LIN {X 0,Y 502.777,Z 286.86,A -85,B 0,C 180,E1 -5904.169,E2 -5904.169} C_VEL
LIN {X 0,Y 502.835,Z 286.849,A -85,B 0,C 180,E1 -5906.993,E2 -5906.993} C_VEL
LIN {X 0,Y 502.818,Z 286.854,A -85,B 0,C 180,E1 -5910.065,E2 -5910.065} C_VEL
LIN {X 0,Y 502.832,Z 286.851,A -85,B 0,C 180,E1 -5912.533,E2 -5912.533} C_VEL
LIN {X 0,Y 502.745,Z 286.865,A -85,B 0,C 180,E1 -5915.32,E2 -5915.32} C_VEL
LIN {X 0,Y 502.634,Z 287.212,A -85,B 0,C 180,E1 -5916.952,E2 -5916.952} C_VEL
LIN {X 0,Y 502.627,Z 289.501,A -85,B 0,C 180,E1 -5919.539,E2 -5919.539} C_VEL
LIN {X 0,Y 502.586,Z 291.79,A -85,B 0,C 180,E1 -5922.083,E2 -5922.083} C_VEL
LIN {X 0,Y 502.483,Z 294.829,A -85,B 0,C 180,E1 -5925.418,E2 -5925.418} C_VEL
LIN {X 0,Y 502.45,Z 295.372,A -85,B 0,C 180,E1 -5925.967,E2 -5925.967} C_VEL
LIN {X 0,Y 504.497,Z 304.103,A -85,B 0,C 180,E1 -5926.262,E2 -5926.262} C_VEL
LIN {X 0,Y 504.385,Z 317.099,A -85,B 0,C 180,E1 -5926.76,E2 -5926.76} C_VEL
LIN {X 0,Y 504.121,Z 329.241,A -85,B 0,C 180,E1 -5927.391,E2 -5927.391} C_VEL
LIN {X 0,Y 503.852,Z 340.243,A -85,B 0,C 180,E1 -5928.127,E2 -5928.127} C_VEL
LIN {X 0,Y 503.535,Z 350.991,A -85,B 0,C 180,E1 -5929.037,E2 -5929.037} C_VEL
LIN {X 0,Y 503.275,Z 359.741,A -85,B 0,C 180,E1 -5929.947,E2 -5929.947} C_VEL
LIN {X 0,Y 503.027,Z 367.754,A -85,B 0,C 180,E1 -5930.957,E2 -5930.957} C_VEL
LIN {X 0,Y 502.758,Z 375.603,A -85,B 0,C 180,E1 -5932.167,E2 -5932.167} C_VEL
LIN {X 0,Y 502.504,Z 382.721,A -85,B 0,C 180,E1 -5933.576,E2 -5933.576} C_VEL
LIN {X 0,Y 502.378,Z 387.441,A -85,B 0,C 180,E1 -5934.783,E2 -5934.783} C_VEL
LIN {X 0,Y 502.368,Z 391.03,A -85,B 0,C 180,E1 -5935.989,E2 -5935.989} C_VEL
LIN {X 0,Y 502.264,Z 392.903,A -85,B 0,C 180,E1 -5936.791,E2 -5936.791} C_VEL
LIN {X 0,Y 502.172,Z 394.318,A -85,B 0,C 180,E1 -5937.594,E2 -5937.594} C_VEL
LIN {X 0,Y 502.095,Z 395.883,A -85,B 0,C 180,E1 -5939.198,E2 -5939.198} C_VEL
LIN {X 0,Y 502.088,Z 396.094,A -85,B 0,C 180,E1 -5940,E2 -5940} C_VEL
LIN {X 0,Y 502.091,Z 395.878,A -85,B 0,C 180,E1 -5940.802,E2 -5940.802} C_VEL
LIN {X 0,Y 502.156,Z 394.273,A -85,B 0,C 180,E1 -5942.406,E2 -5942.406} C_VEL
LIN {X 0,Y 502.257,Z 392.849,A -85,B 0,C 180,E1 -5943.209,E2 -5943.209} C_VEL
LIN {X 0,Y 502.367,Z 389.926,A -85,B 0,C 180,E1 -5944.413,E2 -5944.413} C_VEL
LIN {X 0,Y 502.349,Z 385.983,A -85,B 0,C 180,E1 -5945.62,E2 -5945.62} C_VEL
LIN {X 0,Y 502.56,Z 380.845,A -85,B 0,C 180,E1 -5946.833,E2 -5946.833} C_VEL
LIN {X 0,Y 502.707,Z 374.417,A -85,B 0,C 180,E1 -5948.037,E2 -5948.037} C_VEL
LIN {X 0,Y 502.959,Z 366.358,A -85,B 0,C 180,E1 -5949.247,E2 -5949.247} C_VEL
LIN {X 0,Y 503.228,Z 358.139,A -85,B 0,C 180,E1 -5950.257,E2 -5950.257} C_VEL
LIN {X 0,Y 503.541,Z 348.098,A -85,B 0,C 180,E1 -5951.268,E2 -5951.268} C_VEL
LIN {X 0,Y 503.888,Z 336.424,A -85,B 0,C 180,E1 -5952.198,E2 -5952.198} C_VEL
LIN {X 0,Y 504.152,Z 325.502,A -85,B 0,C 180,E1 -5952.888,E2 -5952.888} C_VEL
LIN {X 0,Y 504.441,Z 314.183,A -85,B 0,C 180,E1 -5953.444,E2 -5953.444} C_VEL
LIN {X 0,Y 504.385,Z 303.242,A -85,B 0,C 180,E1 -5953.856,E2 -5953.856} C_VEL
LIN {X 0,Y 502.24,Z 293.249,A -85,B 0,C 180,E1 -5954.201,E2 -5954.201} C_VEL
LIN {X 0,Y 502.22,Z 290.004,A -85,B 0,C 180,E1 -5957.09,E2 -5957.09} C_VEL
LIN {X 0,Y 502.21,Z 287.179,A -85,B 0,C 180,E1 -5959.625,E2 -5959.625} C_VEL
LIN {X 0,Y 502.509,Z 286.893,A -85,B 0,C 180,E1 -5962.186,E2 -5962.186} C_VEL
LIN {X 0,Y 502.749,Z 286.862,A -85,B 0,C 180,E1 -5964.795,E2 -5964.795} C_VEL
LIN {X 0,Y 502.83,Z 286.845,A -85,B 0,C 180,E1 -5967.467,E2 -5967.467} C_VEL
LIN {X 0,Y 502.811,Z 286.853,A -85,B 0,C 180,E1 -5970.211,E2 -5970.211} C_VEL
LIN {X 0,Y 502.835,Z 286.847,A -85,B 0,C 180,E1 -5973.031,E2 -5973.031} C_VEL
LIN {X 0,Y 502.776,Z 286.855,A -85,B 0,C 180,E1 -5975.951,E2 -5975.951} C_VEL
LIN {X 0,Y 502.805,Z 286.85,A -85,B 0,C 180,E1 -5978.976,E2 -5978.976} C_VEL
LIN {X 0,Y 502.8,Z 286.858,A -85,B 0,C 180,E1 -5982.139,E2 -5982.139} C_VEL
LIN {X 0,Y 502.804,Z 286.852,A -85,B 0,C 180,E1 -5985.468,E2 -5985.468} C_VEL
LIN {X 0,Y 502.823,Z 286.848,A -85,B 0,C 180,E1 -5988.934,E2 -5988.934} C_VEL
LIN {X 0,Y 502.796,Z 286.854,A -85,B 0,C 180,E1 -5992.046,E2 -5992.046} C_VEL
LIN {X 0,Y 502.757,Z 286.857,A -85,B 0,C 180,E1 -5993.311,E2 -5993.311} C_VEL
LIN {X 0,Y 502.063,Z 286.969,A -85,B 0,C 180,E1 -5993.981,E2 -5993.981} C_VEL
LIN {X 0,Y 499.152,Z 287.31,A -85,B 0,C 180,E1 -5995.069,E2 -5995.069} C_VEL
LIN {X 0,Y 496.681,Z 287.621,A -85,B 0,C 180,E1 -5995.941,E2 -5995.941} C_VEL
LIN {X 0,Y 495.581,Z 288.094,A -85,B 0,C 180,E1 -5996.61,E2 -5996.61} C_VEL
LIN {X 0,Y 495.472,Z 288.423,A -85,B 0,C 180,E1 -5996.834,E2 -5996.834} C_VEL
LIN {X 0,Y 495.363,Z 292.704,A -85,B 0,C 180,E1 -5999.286,E2 -5999.286} C_VEL
LIN {X 0,Y 495.342,Z 297.433,A -85,B 0,C 180,E1 -6002.082,E2 -6002.082} C_VEL
LIN {X 0,Y 495.339,Z 302.675,A -85,B 0,C 180,E1 -6005.238,E2 -6005.238} C_VEL
LIN {X 0,Y 495.229,Z 307.861,A -85,B 0,C 180,E1 -6008.347,E2 -6008.347} C_VEL
LIN {X 0,Y 495.203,Z 312.327,A -85,B 0,C 180,E1 -6010.948,E2 -6010.948} C_VEL
LIN {X 0,Y 495.16,Z 316.922,A -85,B 0,C 180,E1 -6013.509,E2 -6013.509} C_VEL
LIN {X 0,Y 495.232,Z 320.815,A -85,B 0,C 180,E1 -6015.581,E2 -6015.581} C_VEL
LIN {X 0,Y 497.789,Z 333.295,A -85,B 0,C 180,E1 -6015.982,E2 -6015.982} C_VEL
LIN {X 0,Y 497.643,Z 345.934,A -85,B 0,C 180,E1 -6016.473,E2 -6016.473} C_VEL
LIN {X 0,Y 497.244,Z 358.46,A -85,B 0,C 180,E1 -6017.141,E2 -6017.141} C_VEL
LIN {X 0,Y 496.901,Z 370.191,A -85,B 0,C 180,E1 -6017.959,E2 -6017.959} C_VEL
LIN {X 0,Y 496.537,Z 380.605,A -85,B 0,C 180,E1 -6018.881,E2 -6018.881} C_VEL
LIN {X 0,Y 496.156,Z 390.869,A -85,B 0,C 180,E1 -6020.007,E2 -6020.007} C_VEL
LIN {X 0,Y 495.79,Z 399.762,A -85,B 0,C 180,E1 -6021.235,E2 -6021.235} C_VEL
LIN {X 0,Y 495.527,Z 406.907,A -85,B 0,C 180,E1 -6022.462,E2 -6022.462} C_VEL
LIN {X 0,Y 495.353,Z 411.752,A -85,B 0,C 180,E1 -6023.483,E2 -6023.483} C_VEL
LIN {X 0,Y 495.141,Z 416.445,A -85,B 0,C 180,E1 -6024.706,E2 -6024.706} C_VEL
LIN {X 0,Y 495.179,Z 420.026,A -85,B 0,C 180,E1 -6025.931,E2 -6025.931} C_VEL
LIN {X 0,Y 495.158,Z 421.873,A -85,B 0,C 180,E1 -6026.745,E2 -6026.745} C_VEL
LIN {X 0,Y 495.064,Z 423.29,A -85,B 0,C 180,E1 -6027.559,E2 -6027.559} C_VEL
LIN {X 0,Y 494.92,Z 424.899,A -85,B 0,C 180,E1 -6029.186,E2 -6029.186} C_VEL
LIN {X 0,Y 494.916,Z 425.136,A -85,B 0,C 180,E1 -6030,E2 -6030} C_VEL
LIN {X 0,Y 494.964,Z 424.371,A -85,B 0,C 180,E1 -6031.627,E2 -6031.627} C_VEL
LIN {X 0,Y 495.158,Z 422.058,A -85,B 0,C 180,E1 -6033.255,E2 -6033.255} C_VEL
LIN {X 0,Y 495.165,Z 419.219,A -85,B 0,C 180,E1 -6034.477,E2 -6034.477} C_VEL
LIN {X 0,Y 495.246,Z 415.36,A -85,B 0,C 180,E1 -6035.701,E2 -6035.701} C_VEL
LIN {X 0,Y 495.413,Z 410.361,A -85,B 0,C 180,E1 -6036.925,E2 -6036.925} C_VEL
LIN {X 0,Y 495.623,Z 404.046,A -85,B 0,C 180,E1 -6038.152,E2 -6038.152} C_VEL
LIN {X 0,Y 495.93,Z 396.197,A -85,B 0,C 180,E1 -6039.379,E2 -6039.379} C_VEL
LIN {X 0,Y 496.263,Z 388.18,A -85,B 0,C 180,E1 -6040.403,E2 -6040.403} C_VEL
LIN {X 0,Y 496.62,Z 378.361,A -85,B 0,C 180,E1 -6041.427,E2 -6041.427} C_VEL
LIN {X 0,Y 496.951,Z 367.1,A -85,B 0,C 180,E1 -6042.366,E2 -6042.366} C_VEL
LIN {X 0,Y 497.291,Z 356.493,A -85,B 0,C 180,E1 -6043.069,E2 -6043.069} C_VEL
LIN {X 0,Y 497.653,Z 344.47,A -85,B 0,C 180,E1 -6043.683,E2 -6043.683} C_VEL
LIN {X 0,Y 497.759,Z 333.262,A -85,B 0,C 180,E1 -6044.11,E2 -6044.11} C_VEL
LIN {X 0,Y 495.244,Z 320.782,A -85,B 0,C 180,E1 -6044.511,E2 -6044.511} C_VEL
LIN {X 0,Y 495.193,Z 314.298,A -85,B 0,C 180,E1 -6048.029,E2 -6048.029} C_VEL
LIN {X 0,Y 495.21,Z 309.511,A -85,B 0,C 180,E1 -6050.781,E2 -6050.781} C_VEL
LIN {X 0,Y 495.272,Z 305.085,A -85,B 0,C 180,E1 -6053.411,E2 -6053.411} C_VEL
LIN {X 0,Y 495.305,Z 300.623,A -85,B 0,C 180,E1 -6056.096,E2 -6056.096} C_VEL
LIN {X 0,Y 495.357,Z 296.067,A -85,B 0,C 180,E1 -6058.841,E2 -6058.841} C_VEL
LIN {X 0,Y 495.435,Z 291.24,A -85,B 0,C 180,E1 -6061.665,E2 -6061.665} C_VEL
LIN {X 0,Y 495.542,Z 287.763,A -85,B 0,C 180,E1 -6063.703,E2 -6063.703} C_VEL
LIN {X 0,Y 495.713,Z 287.74,A -85,B 0,C 180,E1 -6066.087,E2 -6066.087} C_VEL
LIN {X 0,Y 495.766,Z 287.732,A -85,B 0,C 180,E1 -6068.768,E2 -6068.768} C_VEL
LIN {X 0,Y 495.759,Z 287.732,A -85,B 0,C 180,E1 -6071.781,E2 -6071.781} C_VEL
LIN {X 0,Y 495.74,Z 287.737,A -85,B 0,C 180,E1 -6075.141,E2 -6075.141} C_VEL
LIN {X 0,Y 495.759,Z 287.731,A -85,B 0,C 180,E1 -6078.219,E2 -6078.219} C_VEL
LIN {X 0,Y 495.753,Z 287.734,A -85,B 0,C 180,E1 -6081.408,E2 -6081.408} C_VEL
LIN {X 0,Y 495.684,Z 287.74,A -85,B 0,C 180,E1 -6084.457,E2 -6084.457} C_VEL
LIN {X 0,Y 495.498,Z 287.867,A -85,B 0,C 180,E1 -6086.652,E2 -6086.652} C_VEL
LIN {X 0,Y 495.395,Z 292.519,A -85,B 0,C 180,E1 -6089.288,E2 -6089.288} C_VEL
LIN {X 0,Y 495.337,Z 297.457,A -85,B 0,C 180,E1 -6092.081,E2 -6092.081} C_VEL
LIN {X 0,Y 495.352,Z 302.923,A -85,B 0,C 180,E1 -6095.234,E2 -6095.234} C_VEL
LIN {X 0,Y 495.275,Z 308.313,A -85,B 0,C 180,E1 -6098.349,E2 -6098.349} C_VEL
LIN {X 0,Y 495.221,Z 312.805,A -85,B 0,C 180,E1 -6100.949,E2 -6100.949} C_VEL
LIN {X 0,Y 495.191,Z 317.207,A -85,B 0,C 180,E1 -6103.51,E2 -6103.51} C_VEL
LIN {X 0,Y 495.215,Z 321.03,A -85,B 0,C 180,E1 -6105.698,E2 -6105.698} C_VEL
LIN {X 0,Y 497.608,Z 333.51,A -85,B 0,C 180,E1 -6106.107,E2 -6106.107} C_VEL
LIN {X 0,Y 497.316,Z 346.375,A -85,B 0,C 180,E1 -6106.62,E2 -6106.62} C_VEL
LIN {X 0,Y 496.997,Z 358.421,A -85,B 0,C 180,E1 -6107.27,E2 -6107.27} C_VEL
LIN {X 0,Y 496.737,Z 369.713,A -85,B 0,C 180,E1 -6108.058,E2 -6108.058} C_VEL
LIN {X 0,Y 496.369,Z 380.327,A -85,B 0,C 180,E1 -6108.98,E2 -6108.98} C_VEL
LIN {X 0,Y 496.032,Z 389.812,A -85,B 0,C 180,E1 -6110.005,E2 -6110.005} C_VEL
LIN {X 0,Y 495.76,Z 397.6,A -85,B 0,C 180,E1 -6111.029,E2 -6111.029} C_VEL
LIN {X 0,Y 495.515,Z 405.282,A -85,B 0,C 180,E1 -6112.256,E2 -6112.256} C_VEL
LIN {X 0,Y 495.341,Z 411.412,A -85,B 0,C 180,E1 -6113.482,E2 -6113.482} C_VEL
LIN {X 0,Y 495.137,Z 416.249,A -85,B 0,C 180,E1 -6114.706,E2 -6114.706} C_VEL
LIN {X 0,Y 495.177,Z 419.949,A -85,B 0,C 180,E1 -6115.931,E2 -6115.931} C_VEL
LIN {X 0,Y 495.158,Z 421.841,A -85,B 0,C 180,E1 -6116.745,E2 -6116.745} C_VEL
LIN {X 0,Y 495.064,Z 423.311,A -85,B 0,C 180,E1 -6117.559,E2 -6117.559} C_VEL
LIN {X 0,Y 494.966,Z 424.373,A -85,B 0,C 180,E1 -6118.373,E2 -6118.373} C_VEL
LIN {X 0,Y 494.923,Z 425.018,A -85,B 0,C 180,E1 -6119.186,E2 -6119.186} C_VEL
LIN {X 0,Y 494.921,Z 425.259,A -85,B 0,C 180,E1 -6120,E2 -6120} C_VEL
LIN {X 0,Y 494.925,Z 425.103,A -85,B 0,C 180,E1 -6120.814,E2 -6120.814} C_VEL
LIN {X 0,Y 494.967,Z 424.539,A -85,B 0,C 180,E1 -6121.627,E2 -6121.627} C_VEL
LIN {X 0,Y 495.064,Z 423.562,A -85,B 0,C 180,E1 -6122.441,E2 -6122.441} C_VEL
LIN {X 0,Y 495.175,Z 422.178,A -85,B 0,C 180,E1 -6123.255,E2 -6123.255} C_VEL
LIN {X 0,Y 495.17,Z 419.287,A -85,B 0,C 180,E1 -6124.477,E2 -6124.477} C_VEL
LIN {X 0,Y 495.244,Z 415.341,A -85,B 0,C 180,E1 -6125.701,E2 -6125.701} C_VEL
LIN {X 0,Y 495.429,Z 409.348,A -85,B 0,C 180,E1 -6127.11,E2 -6127.11} C_VEL
LIN {X 0,Y 495.619,Z 402.561,A -85,B 0,C 180,E1 -6128.357,E2 -6128.357} C_VEL
LIN {X 0,Y 495.906,Z 394.128,A -85,B 0,C 180,E1 -6129.586,E2 -6129.586} C_VEL
LIN {X 0,Y 496.177,Z 385.491,A -85,B 0,C 180,E1 -6130.611,E2 -6130.611} C_VEL
LIN {X 0,Y 496.548,Z 375.98,A -85,B 0,C 180,E1 -6131.532,E2 -6131.532} C_VEL
LIN {X 0,Y 496.83,Z 364.145,A -85,B 0,C 180,E1 -6132.454,E2 -6132.454} C_VEL
LIN {X 0,Y 497.158,Z 352.181,A -85,B 0,C 180,E1 -6133.176,E2 -6133.176} C_VEL
LIN {X 0,Y 497.488,Z 339.805,A -85,B 0,C 180,E1 -6133.74,E2 -6133.74} C_VEL
LIN {X 0,Y 497.391,Z 332.518,A -85,B 0,C 180,E1 -6134.003,E2 -6134.003} C_VEL
LIN {X 0,Y 495.304,Z 322.078,A -85,B 0,C 180,E1 -6134.351,E2 -6134.351} C_VEL
LIN {X 0,Y 495.29,Z 316.855,A -85,B 0,C 180,E1 -6137.337,E2 -6137.337} C_VEL
LIN {X 0,Y 495.354,Z 310.64,A -85,B 0,C 180,E1 -6140.775,E2 -6140.775} C_VEL
LIN {X 0,Y 495.347,Z 305.658,A -85,B 0,C 180,E1 -6143.407,E2 -6143.407} C_VEL
LIN {X 0,Y 495.289,Z 300.342,A -85,B 0,C 180,E1 -6146.096,E2 -6146.096} C_VEL
LIN {X 0,Y 495.306,Z 294.597,A -85,B 0,C 180,E1 -6148.845,E2 -6148.845} C_VEL
LIN {X 0,Y 495.282,Z 287.796,A -85,B 0,C 180,E1 -6151.79,E2 -6151.79} C_VEL
LIN {X 0,Y 495.729,Z 287.737,A -85,B 0,C 180,E1 -6154.547,E2 -6154.547} C_VEL
LIN {X 0,Y 495.731,Z 287.737,A -85,B 0,C 180,E1 -6157.562,E2 -6157.562} C_VEL
LIN {X 0,Y 495.761,Z 287.732,A -85,B 0,C 180,E1 -6160.047,E2 -6160.047} C_VEL
LIN {X 0,Y 495.719,Z 287.739,A -85,B 0,C 180,E1 -6162.884,E2 -6162.884} C_VEL
LIN {X 0,Y 495.733,Z 287.735,A -85,B 0,C 180,E1 -6165.999,E2 -6165.999} C_VEL
LIN {X 0,Y 495.764,Z 287.734,A -85,B 0,C 180,E1 -6169.3,E2 -6169.3} C_VEL
LIN {X 0,Y 495.784,Z 287.81,A -85,B 0,C 180,E1 -6169.75,E2 -6169.75} C_VEL
LIN {X 0,Y 497.3,Z 295.706,A -85,B 0,C 180,E1 -6172.577,E2 -6172.577} C_VEL
LIN {X 0,Y 497.951,Z 300.349,A -85,B 0,C 180,E1 -6174.146,E2 -6174.146} C_VEL
LIN {X 0,Y 497.582,Z 308.259,A -85,B 0,C 180,E1 -6176.575,E2 -6176.575} C_VEL
LIN {X 0,Y 497.24,Z 318.209,A -85,B 0,C 180,E1 -6179.562,E2 -6179.562} C_VEL
LIN {X 0,Y 496.824,Z 328.593,A -85,B 0,C 180,E1 -6182.63,E2 -6182.63} C_VEL
LIN {X 0,Y 496.528,Z 339.673,A -85,B 0,C 180,E1 -6185.765,E2 -6185.765} C_VEL
LIN {X 0,Y 496.175,Z 350.733,A -85,B 0,C 180,E1 -6188.827,E2 -6188.827} C_VEL
LIN {X 0,Y 495.884,Z 361.475,A -85,B 0,C 180,E1 -6191.832,E2 -6191.832} C_VEL
LIN {X 0,Y 495.547,Z 372.718,A -85,B 0,C 180,E1 -6194.926,E2 -6194.926} C_VEL
LIN {X 0,Y 495.535,Z 374.712,A -85,B 0,C 180,E1 -6195.472,E2 -6195.472} C_VEL
LIN {X 0,Y 497.769,Z 388.179,A -85,B 0,C 180,E1 -6195.851,E2 -6195.851} C_VEL
LIN {X 0,Y 497.547,Z 400.981,A -85,B 0,C 180,E1 -6196.314,E2 -6196.314} C_VEL
LIN {X 0,Y 497.165,Z 413.171,A -85,B 0,C 180,E1 -6196.928,E2 -6196.928} C_VEL
LIN {X 0,Y 496.815,Z 423.896,A -85,B 0,C 180,E1 -6197.625,E2 -6197.625} C_VEL
LIN {X 0,Y 496.472,Z 434.263,A -85,B 0,C 180,E1 -6198.466,E2 -6198.466} C_VEL
LIN {X 0,Y 496.068,Z 443.539,A -85,B 0,C 180,E1 -6199.387,E2 -6199.387} C_VEL
LIN {X 0,Y 495.791,Z 451.992,A -85,B 0,C 180,E1 -6200.412,E2 -6200.412} C_VEL
LIN {X 0,Y 495.485,Z 460.236,A -85,B 0,C 180,E1 -6201.64,E2 -6201.64} C_VEL
LIN {X 0,Y 495.261,Z 466.876,A -85,B 0,C 180,E1 -6202.868,E2 -6202.868} C_VEL
LIN {X 0,Y 495.178,Z 472.95,A -85,B 0,C 180,E1 -6204.298,E2 -6204.298} C_VEL
LIN {X 0,Y 495.029,Z 476.895,A -85,B 0,C 180,E1 -6205.522,E2 -6205.522} C_VEL
LIN {X 0,Y 495.043,Z 479.807,A -85,B 0,C 180,E1 -6206.745,E2 -6206.745} C_VEL
LIN {X 0,Y 494.961,Z 482.183,A -85,B 0,C 180,E1 -6208.373,E2 -6208.373} C_VEL
LIN {X 0,Y 494.898,Z 483,A -85,B 0,C 180,E1 -6210,E2 -6210} C_VEL
LIN {X 0,Y 494.961,Z 482.184,A -85,B 0,C 180,E1 -6211.627,E2 -6211.627} C_VEL
LIN {X 0,Y 495.043,Z 479.81,A -85,B 0,C 180,E1 -6213.255,E2 -6213.255} C_VEL
LIN {X 0,Y 495.029,Z 476.895,A -85,B 0,C 180,E1 -6214.478,E2 -6214.478} C_VEL
LIN {X 0,Y 495.211,Z 471.802,A -85,B 0,C 180,E1 -6215.999,E2 -6215.999} C_VEL
LIN {X 0,Y 495.277,Z 465.869,A -85,B 0,C 180,E1 -6217.337,E2 -6217.337} C_VEL
LIN {X 0,Y 495.557,Z 459.003,A -85,B 0,C 180,E1 -6218.564,E2 -6218.564} C_VEL
LIN {X 0,Y 495.852,Z 450.412,A -85,B 0,C 180,E1 -6219.793,E2 -6219.793} C_VEL
LIN {X 0,Y 496.183,Z 441.598,A -85,B 0,C 180,E1 -6220.817,E2 -6220.817} C_VEL
LIN {X 0,Y 496.58,Z 430.744,A -85,B 0,C 180,E1 -6221.842,E2 -6221.842} C_VEL
LIN {X 0,Y 496.897,Z 420.211,A -85,B 0,C 180,E1 -6222.636,E2 -6222.636} C_VEL
LIN {X 0,Y 497.282,Z 407.499,A -85,B 0,C 180,E1 -6223.381,E2 -6223.381} C_VEL
LIN {X 0,Y 497.7,Z 394.49,A -85,B 0,C 180,E1 -6223.942,E2 -6223.942} C_VEL
LIN {X 0,Y 497.577,Z 386.8,A -85,B 0,C 180,E1 -6224.193,E2 -6224.193} C_VEL
LIN {X 0,Y 495.543,Z 374.64,A -85,B 0,C 180,E1 -6224.548,E2 -6224.548} C_VEL
LIN {X 0,Y 495.856,Z 363.009,A -85,B 0,C 180,E1 -6227.742,E2 -6227.742} C_VEL
LIN {X 0,Y 496.137,Z 352.111,A -85,B 0,C 180,E1 -6230.784,E2 -6230.784} C_VEL
LIN {X 0,Y 496.412,Z 342.767,A -85,B 0,C 180,E1 -6233.354,E2 -6233.354} C_VEL
LIN {X 0,Y 496.673,Z 331.1,A -85,B 0,C 180,E1 -6236.47,E2 -6236.47} C_VEL
LIN {X 0,Y 496.961,Z 319.522,A -85,B 0,C 180,E1 -6239.668,E2 -6239.668} C_VEL
LIN {X 0,Y 497.19,Z 309.679,A -85,B 0,C 180,E1 -6242.49,E2 -6242.49} C_VEL
LIN {X 0,Y 497.493,Z 301.516,A -85,B 0,C 180,E1 -6244.979,E2 -6244.979} C_VEL
LIN {X 0,Y 497.496,Z 297.199,A -85,B 0,C 180,E1 -6246.393,E2 -6246.393} C_VEL
LIN {X 0,Y 496.317,Z 290.614,A -85,B 0,C 180,E1 -6248.847,E2 -6248.847} C_VEL
LIN {X 0,Y 495.744,Z 287.736,A -85,B 0,C 180,E1 -6250.1,E2 -6250.1} C_VEL
LIN {X 0,Y 495.706,Z 287.742,A -85,B 0,C 180,E1 -6252.886,E2 -6252.886} C_VEL
LIN {X 0,Y 495.727,Z 287.737,A -85,B 0,C 180,E1 -6255.998,E2 -6255.998} C_VEL
LIN {X 0,Y 495.742,Z 287.736,A -85,B 0,C 180,E1 -6258.709,E2 -6258.709} C_VEL
LIN {X 0,Y 495.753,Z 287.732,A -85,B 0,C 180,E1 -6261.408,E2 -6261.408} C_VEL
LIN {X 0,Y 495.751,Z 287.734,A -85,B 0,C 180,E1 -6264.462,E2 -6264.462} C_VEL
LIN {X 0,Y 495.77,Z 287.732,A -85,B 0,C 180,E1 -6267.406,E2 -6267.406} C_VEL
LIN {X 0,Y 495.769,Z 287.731,A -85,B 0,C 180,E1 -6270.254,E2 -6270.254} C_VEL
LIN {X 0,Y 495.809,Z 287.729,A -85,B 0,C 180,E1 -6273.255,E2 -6273.255} C_VEL
LIN {X 0,Y 495.656,Z 287.748,A -85,B 0,C 180,E1 -6275.72,E2 -6275.72} C_VEL
LIN {X 0,Y 495.602,Z 287.999,A -85,B 0,C 180,E1 -6276.605,E2 -6276.605} C_VEL
LIN {X 0,Y 495.608,Z 290.421,A -85,B 0,C 180,E1 -6279.377,E2 -6279.377} C_VEL
LIN {X 0,Y 495.547,Z 292.621,A -85,B 0,C 180,E1 -6281.845,E2 -6281.845} C_VEL
LIN {X 0,Y 495.458,Z 295.66,A -85,B 0,C 180,E1 -6285.207,E2 -6285.207} C_VEL
LIN {X 0,Y 495.468,Z 296.302,A -85,B 0,C 180,E1 -6285.784,E2 -6285.784} C_VEL
LIN {X 0,Y 497.681,Z 305.565,A -85,B 0,C 180,E1 -6286.11,E2 -6286.11} C_VEL
LIN {X 0,Y 497.47,Z 318.582,A -85,B 0,C 180,E1 -6286.624,E2 -6286.624} C_VEL
LIN {X 0,Y 497.215,Z 330.124,A -85,B 0,C 180,E1 -6287.239,E2 -6287.239} C_VEL
LIN {X 0,Y 496.941,Z 340.736,A -85,B 0,C 180,E1 -6287.96,E2 -6287.96} C_VEL
LIN {X 0,Y 496.605,Z 351.541,A -85,B 0,C 180,E1 -6288.882,E2 -6288.882} C_VEL
LIN {X 0,Y 496.326,Z 360.324,A -85,B 0,C 180,E1 -6289.805,E2 -6289.805} C_VEL
LIN {X 0,Y 495.998,Z 369.834,A -85,B 0,C 180,E1 -6291.033,E2 -6291.033} C_VEL
LIN {X 0,Y 495.72,Z 377.365,A -85,B 0,C 180,E1 -6292.26,E2 -6292.26} C_VEL
LIN {X 0,Y 495.483,Z 383.385,A -85,B 0,C 180,E1 -6293.484,E2 -6293.484} C_VEL
LIN {X 0,Y 495.354,Z 388.122,A -85,B 0,C 180,E1 -6294.709,E2 -6294.709} C_VEL
LIN {X 0,Y 495.333,Z 391.725,A -85,B 0,C 180,E1 -6295.932,E2 -6295.932} C_VEL
LIN {X 0,Y 495.213,Z 393.594,A -85,B 0,C 180,E1 -6296.746,E2 -6296.746} C_VEL
LIN {X 0,Y 495.112,Z 395.01,A -85,B 0,C 180,E1 -6297.559,E2 -6297.559} C_VEL
LIN {X 0,Y 495.03,Z 396.572,A -85,B 0,C 180,E1 -6299.187,E2 -6299.187} C_VEL
LIN {X 0,Y 495.022,Z 396.778,A -85,B 0,C 180,E1 -6300,E2 -6300} C_VEL
LIN {X 0,Y 495.026,Z 396.565,A -85,B 0,C 180,E1 -6300.814,E2 -6300.814} C_VEL
LIN {X 0,Y 495.092,Z 394.927,A -85,B 0,C 180,E1 -6302.441,E2 -6302.441} C_VEL
LIN {X 0,Y 495.207,Z 393.501,A -85,B 0,C 180,E1 -6303.254,E2 -6303.254} C_VEL
LIN {X 0,Y 495.331,Z 390.553,A -85,B 0,C 180,E1 -6304.476,E2 -6304.476} C_VEL
LIN {X 0,Y 495.307,Z 386.582,A -85,B 0,C 180,E1 -6305.7,E2 -6305.7} C_VEL
LIN {X 0,Y 495.535,Z 380.533,A -85,B 0,C 180,E1 -6307.108,E2 -6307.108} C_VEL
LIN {X 0,Y 495.751,Z 373.703,A -85,B 0,C 180,E1 -6308.355,E2 -6308.355} C_VEL
LIN {X 0,Y 495.991,Z 365.357,A -85,B 0,C 180,E1 -6309.584,E2 -6309.584} C_VEL
LIN {X 0,Y 496.341,Z 356.757,A -85,B 0,C 180,E1 -6310.607,E2 -6310.607} C_VEL
LIN {X 0,Y 496.69,Z 346.13,A -85,B 0,C 180,E1 -6311.633,E2 -6311.633} C_VEL
LIN {X 0,Y 497.022,Z 335.494,A -85,B 0,C 180,E1 -6312.459,E2 -6312.459} C_VEL
LIN {X 0,Y 497.304,Z 323.908,A -85,B 0,C 180,E1 -6313.172,E2 -6313.172} C_VEL
LIN {X 0,Y 497.613,Z 310.599,A -85,B 0,C 180,E1 -6313.788,E2 -6313.788} C_VEL
LIN {X 0,Y 497.471,Z 304.1,A -85,B 0,C 180,E1 -6314.027,E2 -6314.027} C_VEL
LIN {X 0,Y 495.199,Z 293.764,A -85,B 0,C 180,E1 -6314.381,E2 -6314.381} C_VEL
LIN {X 0,Y 495.148,Z 290.426,A -85,B 0,C 180,E1 -6317.342,E2 -6317.342} C_VEL
LIN {X 0,Y 495.159,Z 288.508,A -85,B 0,C 180,E1 -6319.053,E2 -6319.053} C_VEL
LIN {X 0,Y 495.168,Z 287.809,A -85,B 0,C 180,E1 -6319.916,E2 -6319.916} C_VEL
LIN {X 0,Y 495.509,Z 287.765,A -85,B 0,C 180,E1 -6322.791,E2 -6322.791} C_VEL
LIN {X 0,Y 495.719,Z 287.733,A -85,B 0,C 180,E1 -6325.171,E2 -6325.171} C_VEL
LIN {X 0,Y 495.78,Z 287.724,A -85,B 0,C 180,E1 -6327.891,E2 -6327.891} C_VEL
LIN {X 0,Y 495.753,Z 287.73,A -85,B 0,C 180,E1 -6330.687,E2 -6330.687} C_VEL
LIN {X 0,Y 495.762,Z 287.728,A -85,B 0,C 180,E1 -6333.564,E2 -6333.564} C_VEL
LIN {X 0,Y 495.731,Z 287.736,A -85,B 0,C 180,E1 -6336.544,E2 -6336.544} C_VEL
LIN {X 0,Y 495.76,Z 287.729,A -85,B 0,C 180,E1 -6339.638,E2 -6339.638} C_VEL
LIN {X 0,Y 495.741,Z 287.733,A -85,B 0,C 180,E1 -6342.507,E2 -6342.507} C_VEL
LIN {X 0,Y 495.753,Z 287.728,A -85,B 0,C 180,E1 -6345.139,E2 -6345.139} C_VEL
LIN {X 0,Y 495.76,Z 287.73,A -85,B 0,C 180,E1 -6348.219,E2 -6348.219} C_VEL
LIN {X 0,Y 495.753,Z 287.734,A -85,B 0,C 180,E1 -6351.408,E2 -6351.408} C_VEL
LIN {X 0,Y 495.713,Z 287.736,A -85,B 0,C 180,E1 -6354.459,E2 -6354.459} C_VEL
LIN {X 0,Y 495.539,Z 287.88,A -85,B 0,C 180,E1 -6356.536,E2 -6356.536} C_VEL
LIN {X 0,Y 495.472,Z 288.423,A -85,B 0,C 180,E1 -6356.834,E2 -6356.834} C_VEL
LIN {X 0,Y 494.742,Z 289.665,A -85,B 0,C 180,E1 -6357.497,E2 -6357.497} C_VEL
LIN {X 0,Y 491.823,Z 291.856,A -85,B 0,C 180,E1 -6358.567,E2 -6358.567} C_VEL
LIN {X 0,Y 489.391,Z 293.605,A -85,B 0,C 180,E1 -6359.43,E2 -6359.43} C_VEL
LIN {X 0,Y 488.357,Z 294.856,A -85,B 0,C 180,E1 -6360.099,E2 -6360.099} C_VEL
LIN {X 0,Y 488.276,Z 295.241,A -85,B 0,C 180,E1 -6360.327,E2 -6360.327} C_VEL
LIN {X 0,Y 488.257,Z 298.982,A -85,B 0,C 180,E1 -6362.573,E2 -6362.573} C_VEL
LIN {X 0,Y 488.272,Z 303.531,A -85,B 0,C 180,E1 -6365.328,E2 -6365.328} C_VEL
LIN {X 0,Y 488.168,Z 308.009,A -85,B 0,C 180,E1 -6368.018,E2 -6368.018} C_VEL
LIN {X 0,Y 488.133,Z 312.516,A -85,B 0,C 180,E1 -6370.661,E2 -6370.661} C_VEL
LIN {X 0,Y 488.096,Z 317.167,A -85,B 0,C 180,E1 -6373.263,E2 -6373.263} C_VEL
LIN {X 0,Y 488.184,Z 321.174,A -85,B 0,C 180,E1 -6375.368,E2 -6375.368} C_VEL
LIN {X 0,Y 490.953,Z 334.514,A -85,B 0,C 180,E1 -6375.81,E2 -6375.81} C_VEL
LIN {X 0,Y 490.715,Z 347.401,A -85,B 0,C 180,E1 -6376.331,E2 -6376.331} C_VEL
LIN {X 0,Y 490.337,Z 359.136,A -85,B 0,C 180,E1 -6376.974,E2 -6376.974} C_VEL
LIN {X 0,Y 489.975,Z 370.601,A -85,B 0,C 180,E1 -6377.786,E2 -6377.786} C_VEL
LIN {X 0,Y 489.594,Z 381.016,A -85,B 0,C 180,E1 -6378.721,E2 -6378.721} C_VEL
LIN {X 0,Y 489.188,Z 391.281,A -85,B 0,C 180,E1 -6379.864,E2 -6379.864} C_VEL
LIN {X 0,Y 488.791,Z 400.175,A -85,B 0,C 180,E1 -6381.108,E2 -6381.108} C_VEL
LIN {X 0,Y 488.512,Z 407.32,A -85,B 0,C 180,E1 -6382.353,E2 -6382.353} C_VEL
LIN {X 0,Y 488.311,Z 412.166,A -85,B 0,C 180,E1 -6383.388,E2 -6383.388} C_VEL
LIN {X 0,Y 488.085,Z 416.86,A -85,B 0,C 180,E1 -6384.63,E2 -6384.63} C_VEL
LIN {X 0,Y 488.12,Z 420.44,A -85,B 0,C 180,E1 -6385.872,E2 -6385.872} C_VEL
LIN {X 0,Y 488.077,Z 422.289,A -85,B 0,C 180,E1 -6386.698,E2 -6386.698} C_VEL
LIN {X 0,Y 488.003,Z 423.704,A -85,B 0,C 180,E1 -6387.524,E2 -6387.524} C_VEL
LIN {X 0,Y 487.842,Z 425.314,A -85,B 0,C 180,E1 -6389.175,E2 -6389.175} C_VEL
LIN {X 0,Y 487.836,Z 425.55,A -85,B 0,C 180,E1 -6390,E2 -6390} C_VEL
LIN {X 0,Y 487.894,Z 424.784,A -85,B 0,C 180,E1 -6391.651,E2 -6391.651} C_VEL
LIN {X 0,Y 488.003,Z 423.822,A -85,B 0,C 180,E1 -6392.476,E2 -6392.476} C_VEL
LIN {X 0,Y 488.076,Z 422.471,A -85,B 0,C 180,E1 -6393.302,E2 -6393.302} C_VEL
LIN {X 0,Y 488.099,Z 419.631,A -85,B 0,C 180,E1 -6394.542,E2 -6394.542} C_VEL
LIN {X 0,Y 488.199,Z 415.769,A -85,B 0,C 180,E1 -6395.784,E2 -6395.784} C_VEL
LIN {X 0,Y 488.381,Z 410.769,A -85,B 0,C 180,E1 -6397.026,E2 -6397.026} C_VEL
LIN {X 0,Y 488.593,Z 404.453,A -85,B 0,C 180,E1 -6398.27,E2 -6398.27} C_VEL
LIN {X 0,Y 488.925,Z 396.601,A -85,B 0,C 180,E1 -6399.515,E2 -6399.515} C_VEL
LIN {X 0,Y 489.31,Z 388.58,A -85,B 0,C 180,E1 -6400.552,E2 -6400.552} C_VEL
LIN {X 0,Y 489.676,Z 378.758,A -85,B 0,C 180,E1 -6401.592,E2 -6401.592} C_VEL
LIN {X 0,Y 490.03,Z 367.68,A -85,B 0,C 180,E1 -6402.529,E2 -6402.529} C_VEL
LIN {X 0,Y 490.414,Z 356.878,A -85,B 0,C 180,E1 -6403.255,E2 -6403.255} C_VEL
LIN {X 0,Y 490.79,Z 344.838,A -85,B 0,C 180,E1 -6403.878,E2 -6403.878} C_VEL
LIN {X 0,Y 490.837,Z 334.028,A -85,B 0,C 180,E1 -6404.3,E2 -6404.3} C_VEL
LIN {X 0,Y 488.189,Z 321.092,A -85,B 0,C 180,E1 -6404.725,E2 -6404.725} C_VEL
LIN {X 0,Y 488.116,Z 314.784,A -85,B 0,C 180,E1 -6408.142,E2 -6408.142} C_VEL
LIN {X 0,Y 488.162,Z 309.67,A -85,B 0,C 180,E1 -6411.095,E2 -6411.095} C_VEL
LIN {X 0,Y 488.214,Z 305.189,A -85,B 0,C 180,E1 -6413.77,E2 -6413.77} C_VEL
LIN {X 0,Y 488.273,Z 300.671,A -85,B 0,C 180,E1 -6416.5,E2 -6416.5} C_VEL
LIN {X 0,Y 488.288,Z 296.043,A -85,B 0,C 180,E1 -6419.299,E2 -6419.299} C_VEL
LIN {X 0,Y 488.37,Z 291.119,A -85,B 0,C 180,E1 -6422.172,E2 -6422.172} C_VEL
LIN {X 0,Y 488.48,Z 288.643,A -85,B 0,C 180,E1 -6423.6,E2 -6423.6} C_VEL
LIN {X 0,Y 488.67,Z 288.617,A -85,B 0,C 180,E1 -6426.133,E2 -6426.133} C_VEL
LIN {X 0,Y 488.704,Z 288.611,A -85,B 0,C 180,E1 -6429.254,E2 -6429.254} C_VEL
LIN {X 0,Y 488.71,Z 288.61,A -85,B 0,C 180,E1 -6431.6,E2 -6431.6} C_VEL
LIN {X 0,Y 488.704,Z 288.613,A -85,B 0,C 180,E1 -6434.803,E2 -6434.803} C_VEL
LIN {X 0,Y 488.694,Z 288.615,A -85,B 0,C 180,E1 -6437.474,E2 -6437.474} C_VEL
LIN {X 0,Y 488.736,Z 288.606,A -85,B 0,C 180,E1 -6439.677,E2 -6439.677} C_VEL
LIN {X 0,Y 488.672,Z 288.617,A -85,B 0,C 180,E1 -6442.84,E2 -6442.84} C_VEL
LIN {X 0,Y 488.546,Z 288.631,A -85,B 0,C 180,E1 -6445.872,E2 -6445.872} C_VEL
LIN {X 0,Y 488.419,Z 288.817,A -85,B 0,C 180,E1 -6446.746,E2 -6446.746} C_VEL
LIN {X 0,Y 488.336,Z 294.116,A -85,B 0,C 180,E1 -6449.754,E2 -6449.754} C_VEL
LIN {X 0,Y 488.256,Z 299.044,A -85,B 0,C 180,E1 -6452.573,E2 -6452.573} C_VEL
LIN {X 0,Y 488.288,Z 303.819,A -85,B 0,C 180,E1 -6455.329,E2 -6455.329} C_VEL
LIN {X 0,Y 488.201,Z 308.445,A -85,B 0,C 180,E1 -6458.02,E2 -6458.02} C_VEL
LIN {X 0,Y 488.161,Z 312.971,A -85,B 0,C 180,E1 -6460.663,E2 -6460.663} C_VEL
LIN {X 0,Y 488.123,Z 317.451,A -85,B 0,C 180,E1 -6463.264,E2 -6463.264} C_VEL
LIN {X 0,Y 488.172,Z 321.316,A -85,B 0,C 180,E1 -6465.501,E2 -6465.501} C_VEL
LIN {X 0,Y 490.69,Z 334.833,A -85,B 0,C 180,E1 -6465.96,E2 -6465.96} C_VEL
LIN {X 0,Y 490.371,Z 347.453,A -85,B 0,C 180,E1 -6466.48,E2 -6466.48} C_VEL
LIN {X 0,Y 490.026,Z 359.513,A -85,B 0,C 180,E1 -6467.152,E2 -6467.152} C_VEL
LIN {X 0,Y 489.76,Z 371.161,A -85,B 0,C 180,E1 -6467.99,E2 -6467.99} C_VEL
LIN {X 0,Y 489.364,Z 381.543,A -85,B 0,C 180,E1 -6468.925,E2 -6468.925} C_VEL
LIN {X 0,Y 488.967,Z 391.761,A -85,B 0,C 180,E1 -6470.068,E2 -6470.068} C_VEL
LIN {X 0,Y 488.637,Z 400.661,A -85,B 0,C 180,E1 -6471.314,E2 -6471.314} C_VEL
LIN {X 0,Y 488.421,Z 407.805,A -85,B 0,C 180,E1 -6472.559,E2 -6472.559} C_VEL
LIN {X 0,Y 488.276,Z 413.524,A -85,B 0,C 180,E1 -6473.803,E2 -6473.803} C_VEL
LIN {X 0,Y 488.036,Z 417.997,A -85,B 0,C 180,E1 -6475.043,E2 -6475.043} C_VEL
LIN {X 0,Y 488.116,Z 420.344,A -85,B 0,C 180,E1 -6475.872,E2 -6475.872} C_VEL
LIN {X 0,Y 488.076,Z 422.254,A -85,B 0,C 180,E1 -6476.698,E2 -6476.698} C_VEL
LIN {X 0,Y 488.003,Z 423.743,A -85,B 0,C 180,E1 -6477.524,E2 -6477.524} C_VEL
LIN {X 0,Y 487.895,Z 424.801,A -85,B 0,C 180,E1 -6478.349,E2 -6478.349} C_VEL
LIN {X 0,Y 487.841,Z 425.713,A -85,B 0,C 180,E1 -6480,E2 -6480} C_VEL
LIN {X 0,Y 487.847,Z 425.549,A -85,B 0,C 180,E1 -6480.825,E2 -6480.825} C_VEL
LIN {X 0,Y 488.004,Z 424.015,A -85,B 0,C 180,E1 -6482.476,E2 -6482.476} C_VEL
LIN {X 0,Y 488.105,Z 422.62,A -85,B 0,C 180,E1 -6483.302,E2 -6483.302} C_VEL
LIN {X 0,Y 488.106,Z 419.721,A -85,B 0,C 180,E1 -6484.542,E2 -6484.542} C_VEL
LIN {X 0,Y 488.196,Z 415.756,A -85,B 0,C 180,E1 -6485.784,E2 -6485.784} C_VEL
LIN {X 0,Y 488.393,Z 409.743,A -85,B 0,C 180,E1 -6487.213,E2 -6487.213} C_VEL
LIN {X 0,Y 488.618,Z 402.913,A -85,B 0,C 180,E1 -6488.478,E2 -6488.478} C_VEL
LIN {X 0,Y 488.911,Z 394.456,A -85,B 0,C 180,E1 -6489.724,E2 -6489.724} C_VEL
LIN {X 0,Y 489.202,Z 385.785,A -85,B 0,C 180,E1 -6490.764,E2 -6490.764} C_VEL
LIN {X 0,Y 489.658,Z 375.001,A -85,B 0,C 180,E1 -6491.802,E2 -6491.802} C_VEL
LIN {X 0,Y 489.899,Z 364.059,A -85,B 0,C 180,E1 -6492.652,E2 -6492.652} C_VEL
LIN {X 0,Y 490.231,Z 352.225,A -85,B 0,C 180,E1 -6493.366,E2 -6493.366} C_VEL
LIN {X 0,Y 490.579,Z 339.754,A -85,B 0,C 180,E1 -6493.937,E2 -6493.937} C_VEL
LIN {X 0,Y 490.507,Z 333.579,A -85,B 0,C 180,E1 -6494.164,E2 -6494.164} C_VEL
LIN {X 0,Y 488.264,Z 322.565,A -85,B 0,C 180,E1 -6494.556,E2 -6494.556} C_VEL
LIN {X 0,Y 488.283,Z 316.122,A -85,B 0,C 180,E1 -6498.202,E2 -6498.202} C_VEL
LIN {X 0,Y 488.286,Z 310.876,A -85,B 0,C 180,E1 -6501.09,E2 -6501.09} C_VEL
LIN {X 0,Y 488.288,Z 305.821,A -85,B 0,C 180,E1 -6503.766,E2 -6503.766} C_VEL
LIN {X 0,Y 488.239,Z 299.717,A -85,B 0,C 180,E1 -6506.815,E2 -6506.815} C_VEL
LIN {X 0,Y 488.266,Z 296.044,A -85,B 0,C 180,E1 -6508.595,E2 -6508.595} C_VEL
LIN {X 0,Y 488.237,Z 288.673,A -85,B 0,C 180,E1 -6511.793,E2 -6511.793} C_VEL
LIN {X 0,Y 488.613,Z 288.625,A -85,B 0,C 180,E1 -6514.122,E2 -6514.122} C_VEL
LIN {X 0,Y 488.683,Z 288.616,A -85,B 0,C 180,E1 -6516.354,E2 -6516.354} C_VEL
LIN {X 0,Y 488.703,Z 288.612,A -85,B 0,C 180,E1 -6519.254,E2 -6519.254} C_VEL
LIN {X 0,Y 488.69,Z 288.613,A -85,B 0,C 180,E1 -6522.526,E2 -6522.526} C_VEL
LIN {X 0,Y 488.714,Z 288.61,A -85,B 0,C 180,E1 -6525.199,E2 -6525.199} C_VEL
LIN {X 0,Y 488.697,Z 288.614,A -85,B 0,C 180,E1 -6528.583,E2 -6528.583} C_VEL
LIN {X 0,Y 488.725,Z 288.663,A -85,B 0,C 180,E1 -6529.405,E2 -6529.405} C_VEL
LIN {X 0,Y 490.156,Z 295.946,A -85,B 0,C 180,E1 -6532.056,E2 -6532.056} C_VEL
LIN {X 0,Y 491.017,Z 301.689,A -85,B 0,C 180,E1 -6534.067,E2 -6534.067} C_VEL
LIN {X 0,Y 490.61,Z 309.791,A -85,B 0,C 180,E1 -6536.589,E2 -6536.589} C_VEL
LIN {X 0,Y 490.284,Z 318.772,A -85,B 0,C 180,E1 -6539.325,E2 -6539.325} C_VEL
LIN {X 0,Y 489.842,Z 328.327,A -85,B 0,C 180,E1 -6542.206,E2 -6542.206} C_VEL
LIN {X 0,Y 489.544,Z 338.165,A -85,B 0,C 180,E1 -6545.074,E2 -6545.074} C_VEL
LIN {X 0,Y 489.222,Z 348.931,A -85,B 0,C 180,E1 -6548.068,E2 -6548.068} C_VEL
LIN {X 0,Y 488.895,Z 359.94,A -85,B 0,C 180,E1 -6551.129,E2 -6551.129} C_VEL
LIN {X 0,Y 488.587,Z 370.683,A -85,B 0,C 180,E1 -6554.139,E2 -6554.139} C_VEL
LIN {X 0,Y 488.491,Z 374.712,A -85,B 0,C 180,E1 -6555.258,E2 -6555.258} C_VEL
LIN {X 0,Y 490.813,Z 388.637,A -85,B 0,C 180,E1 -6555.66,E2 -6555.66} C_VEL
LIN {X 0,Y 490.662,Z 400.98,A -85,B 0,C 180,E1 -6556.118,E2 -6556.118} C_VEL
LIN {X 0,Y 490.229,Z 413.171,A -85,B 0,C 180,E1 -6556.739,E2 -6556.739} C_VEL
LIN {X 0,Y 489.837,Z 423.895,A -85,B 0,C 180,E1 -6557.446,E2 -6557.446} C_VEL
LIN {X 0,Y 489.498,Z 434.264,A -85,B 0,C 180,E1 -6558.299,E2 -6558.299} C_VEL
LIN {X 0,Y 489.076,Z 443.539,A -85,B 0,C 180,E1 -6559.233,E2 -6559.233} C_VEL
LIN {X 0,Y 488.764,Z 451.992,A -85,B 0,C 180,E1 -6560.273,E2 -6560.273} C_VEL
LIN {X 0,Y 488.454,Z 460.235,A -85,B 0,C 180,E1 -6561.519,E2 -6561.519} C_VEL
LIN {X 0,Y 488.186,Z 466.875,A -85,B 0,C 180,E1 -6562.763,E2 -6562.763} C_VEL
LIN {X 0,Y 488.104,Z 472.95,A -85,B 0,C 180,E1 -6564.215,E2 -6564.215} C_VEL
LIN {X 0,Y 487.938,Z 476.895,A -85,B 0,C 180,E1 -6565.456,E2 -6565.456} C_VEL
LIN {X 0,Y 487.966,Z 479.807,A -85,B 0,C 180,E1 -6566.697,E2 -6566.697} C_VEL
LIN {X 0,Y 487.889,Z 482.183,A -85,B 0,C 180,E1 -6568.349,E2 -6568.349} C_VEL
LIN {X 0,Y 487.819,Z 483,A -85,B 0,C 180,E1 -6570,E2 -6570} C_VEL
LIN {X 0,Y 487.889,Z 482.184,A -85,B 0,C 180,E1 -6571.651,E2 -6571.651} C_VEL
LIN {X 0,Y 487.966,Z 479.81,A -85,B 0,C 180,E1 -6573.303,E2 -6573.303} C_VEL
LIN {X 0,Y 487.938,Z 476.895,A -85,B 0,C 180,E1 -6574.544,E2 -6574.544} C_VEL
LIN {X 0,Y 488.105,Z 472.948,A -85,B 0,C 180,E1 -6575.785,E2 -6575.785} C_VEL
LIN {X 0,Y 488.19,Z 466.875,A -85,B 0,C 180,E1 -6577.237,E2 -6577.237} C_VEL
LIN {X 0,Y 488.454,Z 460.235,A -85,B 0,C 180,E1 -6578.481,E2 -6578.481} C_VEL
LIN {X 0,Y 488.764,Z 451.991,A -85,B 0,C 180,E1 -6579.727,E2 -6579.727} C_VEL
LIN {X 0,Y 489.077,Z 443.539,A -85,B 0,C 180,E1 -6580.767,E2 -6580.767} C_VEL
LIN {X 0,Y 489.568,Z 433.092,A -85,B 0,C 180,E1 -6581.804,E2 -6581.804} C_VEL
LIN {X 0,Y 489.893,Z 421.886,A -85,B 0,C 180,E1 -6582.701,E2 -6582.701} C_VEL
LIN {X 0,Y 490.246,Z 411.404,A -85,B 0,C 180,E1 -6583.366,E2 -6583.366} C_VEL
LIN {X 0,Y 490.681,Z 399.762,A -85,B 0,C 180,E1 -6583.934,E2 -6583.934} C_VEL
LIN {X 0,Y 490.775,Z 388.171,A -85,B 0,C 180,E1 -6584.354,E2 -6584.354} C_VEL
LIN {X 0,Y 488.482,Z 374.64,A -85,B 0,C 180,E1 -6584.763,E2 -6584.763} C_VEL
LIN {X 0,Y 488.831,Z 363.071,A -85,B 0,C 180,E1 -6587.988,E2 -6587.988} C_VEL
LIN {X 0,Y 489.096,Z 352.499,A -85,B 0,C 180,E1 -6590.931,E2 -6590.931} C_VEL
LIN {X 0,Y 489.419,Z 340.407,A -85,B 0,C 180,E1 -6594.158,E2 -6594.158} C_VEL
LIN {X 0,Y 489.678,Z 328.829,A -85,B 0,C 180,E1 -6597.34,E2 -6597.34} C_VEL
LIN {X 0,Y 489.977,Z 318.939,A -85,B 0,C 180,E1 -6600.134,E2 -6600.134} C_VEL
LIN {X 0,Y 490.263,Z 309.231,A -85,B 0,C 180,E1 -6603.007,E2 -6603.007} C_VEL
LIN {X 0,Y 490.551,Z 302.117,A -85,B 0,C 180,E1 -6605.251,E2 -6605.251} C_VEL
LIN {X 0,Y 490.451,Z 298.075,A -85,B 0,C 180,E1 -6606.634,E2 -6606.634} C_VEL
LIN {X 0,Y 489.241,Z 291.487,A -85,B 0,C 180,E1 -6609.203,E2 -6609.203} C_VEL
LIN {X 0,Y 488.682,Z 288.616,A -85,B 0,C 180,E1 -6610.487,E2 -6610.487} C_VEL
LIN {X 0,Y 488.676,Z 288.615,A -85,B 0,C 180,E1 -6613.656,E2 -6613.656} C_VEL
LIN {X 0,Y 488.68,Z 288.616,A -85,B 0,C 180,E1 -6616.345,E2 -6616.345} C_VEL
LIN {X 0,Y 488.72,Z 288.609,A -85,B 0,C 180,E1 -6619.675,E2 -6619.675} C_VEL
LIN {X 0,Y 488.682,Z 288.613,A -85,B 0,C 180,E1 -6622.841,E2 -6622.841} C_VEL
LIN {X 0,Y 488.733,Z 288.609,A -85,B 0,C 180,E1 -6625.887,E2 -6625.887} C_VEL
LIN {X 0,Y 488.695,Z 288.611,A -85,B 0,C 180,E1 -6628.82,E2 -6628.82} C_VEL
LIN {X 0,Y 488.747,Z 288.608,A -85,B 0,C 180,E1 -6631.671,E2 -6631.671} C_VEL
LIN {X 0,Y 488.704,Z 288.612,A -85,B 0,C 180,E1 -6634.442,E2 -6634.442} C_VEL
LIN {X 0,Y 488.577,Z 288.798,A -85,B 0,C 180,E1 -6636.248,E2 -6636.248} C_VEL
LIN {X 0,Y 488.592,Z 291.373,A -85,B 0,C 180,E1 -6639.224,E2 -6639.224} C_VEL
LIN {X 0,Y 488.531,Z 293.552,A -85,B 0,C 180,E1 -6641.71,E2 -6641.71} C_VEL
LIN {X 0,Y 488.448,Z 296.495,A -85,B 0,C 180,E1 -6644.99,E2 -6644.99} C_VEL
LIN {X 0,Y 488.444,Z 297.075,A -85,B 0,C 180,E1 -6645.586,E2 -6645.586} C_VEL
LIN {X 0,Y 490.827,Z 306.627,A -85,B 0,C 180,E1 -6645.938,E2 -6645.938} C_VEL
LIN {X 0,Y 490.595,Z 318.952,A -85,B 0,C 180,E1 -6646.433,E2 -6646.433} C_VEL
LIN {X 0,Y 490.302,Z 331.107,A -85,B 0,C 180,E1 -6647.089,E2 -6647.089} C_VEL
LIN {X 0,Y 489.971,Z 342.582,A -85,B 0,C 180,E1 -6647.891,E2 -6647.891} C_VEL
LIN {X 0,Y 489.629,Z 353.172,A -85,B 0,C 180,E1 -6648.827,E2 -6648.827} C_VEL
LIN {X 0,Y 489.286,Z 362.699,A -85,B 0,C 180,E1 -6649.866,E2 -6649.866} C_VEL
LIN {X 0,Y 489.03,Z 370.476,A -85,B 0,C 180,E1 -6650.904,E2 -6650.904} C_VEL
LIN {X 0,Y 488.722,Z 378.028,A -85,B 0,C 180,E1 -6652.148,E2 -6652.148} C_VEL
LIN {X 0,Y 488.486,Z 384.059,A -85,B 0,C 180,E1 -6653.391,E2 -6653.391} C_VEL
LIN {X 0,Y 488.33,Z 388.808,A -85,B 0,C 180,E1 -6654.632,E2 -6654.632} C_VEL
LIN {X 0,Y 488.299,Z 392.42,A -85,B 0,C 180,E1 -6655.873,E2 -6655.873} C_VEL
LIN {X 0,Y 488.165,Z 394.281,A -85,B 0,C 180,E1 -6656.699,E2 -6656.699} C_VEL
LIN {X 0,Y 488.052,Z 395.7,A -85,B 0,C 180,E1 -6657.524,E2 -6657.524} C_VEL
LIN {X 0,Y 487.965,Z 397.261,A -85,B 0,C 180,E1 -6659.175,E2 -6659.175} C_VEL
LIN {X 0,Y 487.955,Z 397.462,A -85,B 0,C 180,E1 -6660,E2 -6660} C_VEL
LIN {X 0,Y 487.959,Z 397.241,A -85,B 0,C 180,E1 -6660.825,E2 -6660.825} C_VEL
LIN {X 0,Y 488.03,Z 395.582,A -85,B 0,C 180,E1 -6662.476,E2 -6662.476} C_VEL
LIN {X 0,Y 488.159,Z 394.153,A -85,B 0,C 180,E1 -6663.301,E2 -6663.301} C_VEL
LIN {X 0,Y 488.296,Z 391.179,A -85,B 0,C 180,E1 -6664.54,E2 -6664.54} C_VEL
LIN {X 0,Y 488.266,Z 387.182,A -85,B 0,C 180,E1 -6665.783,E2 -6665.783} C_VEL
LIN {X 0,Y 488.509,Z 381.195,A -85,B 0,C 180,E1 -6667.19,E2 -6667.19} C_VEL
LIN {X 0,Y 488.757,Z 374.231,A -85,B 0,C 180,E1 -6668.476,E2 -6668.476} C_VEL
LIN {X 0,Y 489.001,Z 365.844,A -85,B 0,C 180,E1 -6669.722,E2 -6669.722} C_VEL
LIN {X 0,Y 489.387,Z 357.175,A -85,B 0,C 180,E1 -6670.76,E2 -6670.76} C_VEL
LIN {X 0,Y 489.745,Z 346.502,A -85,B 0,C 180,E1 -6671.8,E2 -6671.8} C_VEL
LIN {X 0,Y 490.097,Z 335.821,A -85,B 0,C 180,E1 -6672.638,E2 -6672.638} C_VEL
LIN {X 0,Y 490.393,Z 324.127,A -85,B 0,C 180,E1 -6673.362,E2 -6673.362} C_VEL
LIN {X 0,Y 490.724,Z 310.724,A -85,B 0,C 180,E1 -6673.986,E2 -6673.986} C_VEL
LIN {X 0,Y 490.541,Z 304.954,A -85,B 0,C 180,E1 -6674.203,E2 -6674.203} C_VEL
LIN {X 0,Y 488.139,Z 294.293,A -85,B 0,C 180,E1 -6674.593,E2 -6674.593} C_VEL
LIN {X 0,Y 488.105,Z 290.874,A -85,B 0,C 180,E1 -6677.6,E2 -6677.6} C_VEL
LIN {X 0,Y 488.099,Z 288.885,A -85,B 0,C 180,E1 -6679.34,E2 -6679.34} C_VEL
LIN {X 0,Y 488.377,Z 288.652,A -85,B 0,C 180,E1 -6681.972,E2 -6681.972} C_VEL
LIN {X 0,Y 488.688,Z 288.61,A -85,B 0,C 180,E1 -6685.038,E2 -6685.038} C_VEL
LIN {X 0,Y 488.735,Z 288.601,A -85,B 0,C 180,E1 -6687.398,E2 -6687.398} C_VEL
LIN {X 0,Y 488.712,Z 288.611,A -85,B 0,C 180,E1 -6690.363,E2 -6690.363} C_VEL
LIN {X 0,Y 488.737,Z 288.603,A -85,B 0,C 180,E1 -6693.484,E2 -6693.484} C_VEL
LIN {X 0,Y 488.685,Z 288.617,A -85,B 0,C 180,E1 -6696.355,E2 -6696.355} C_VEL
LIN {X 0,Y 488.704,Z 288.606,A -85,B 0,C 180,E1 -6699.254,E2 -6699.254} C_VEL
LIN {X 0,Y 488.711,Z 288.609,A -85,B 0,C 180,E1 -6701.6,E2 -6701.6} C_VEL
LIN {X 0,Y 488.715,Z 288.605,A -85,B 0,C 180,E1 -6704.801,E2 -6704.801} C_VEL
LIN {X 0,Y 488.695,Z 288.61,A -85,B 0,C 180,E1 -6707.475,E2 -6707.475} C_VEL
LIN {X 0,Y 488.736,Z 288.61,A -85,B 0,C 180,E1 -6709.677,E2 -6709.677} C_VEL
LIN {X 0,Y 488.681,Z 288.61,A -85,B 0,C 180,E1 -6712.841,E2 -6712.841} C_VEL
LIN {X 0,Y 488.556,Z 288.634,A -85,B 0,C 180,E1 -6715.873,E2 -6715.873} C_VEL
LIN {X 0,Y 488.49,Z 288.701,A -85,B 0,C 180,E1 -6716.56,E2 -6716.56} C_VEL
LIN {X 0,Y 488.297,Z 294.273,A -85,B 0,C 180,E1 -6719.751,E2 -6719.751} C_VEL
LIN {X 0,Y 488.276,Z 295.241,A -85,B 0,C 180,E1 -6720.327,E2 -6720.327} C_VEL
LIN {X 0,Y 487.609,Z 296.444,A -85,B 0,C 180,E1 -6721,E2 -6721} C_VEL
LIN {X 0,Y 484.721,Z 298.562,A -85,B 0,C 180,E1 -6722.09,E2 -6722.09} C_VEL
LIN {X 0,Y 482.282,Z 300.263,A -85,B 0,C 180,E1 -6722.967,E2 -6722.967} C_VEL
LIN {X 0,Y 481.248,Z 301.489,A -85,B 0,C 180,E1 -6723.648,E2 -6723.648} C_VEL
LIN {X 0,Y 481.171,Z 301.878,A -85,B 0,C 180,E1 -6723.879,E2 -6723.879} C_VEL
LIN {X 0,Y 481.153,Z 306.639,A -85,B 0,C 180,E1 -6726.773,E2 -6726.773} C_VEL
LIN {X 0,Y 481.083,Z 311.19,A -85,B 0,C 180,E1 -6729.475,E2 -6729.475} C_VEL
LIN {X 0,Y 481.068,Z 315.829,A -85,B 0,C 180,E1 -6732.134,E2 -6732.134} C_VEL
LIN {X 0,Y 481.128,Z 321.532,A -85,B 0,C 180,E1 -6735.149,E2 -6735.149} C_VEL
LIN {X 0,Y 484.009,Z 334.9,A -85,B 0,C 180,E1 -6735.602,E2 -6735.602} C_VEL
LIN {X 0,Y 483.878,Z 346.731,A -85,B 0,C 180,E1 -6736.08,E2 -6736.08} C_VEL
LIN {X 0,Y 483.487,Z 358.408,A -85,B 0,C 180,E1 -6736.714,E2 -6736.714} C_VEL
LIN {X 0,Y 483.098,Z 369.662,A -85,B 0,C 180,E1 -6737.502,E2 -6737.502} C_VEL
LIN {X 0,Y 482.702,Z 380.394,A -85,B 0,C 180,E1 -6738.452,E2 -6738.452} C_VEL
LIN {X 0,Y 482.262,Z 389.969,A -85,B 0,C 180,E1 -6739.504,E2 -6739.504} C_VEL
LIN {X 0,Y 481.918,Z 397.835,A -85,B 0,C 180,E1 -6740.557,E2 -6740.557} C_VEL
LIN {X 0,Y 481.568,Z 405.55,A -85,B 0,C 180,E1 -6741.82,E2 -6741.82} C_VEL
LIN {X 0,Y 481.286,Z 412.225,A -85,B 0,C 180,E1 -6743.206,E2 -6743.206} C_VEL
LIN {X 0,Y 481.033,Z 417.274,A -85,B 0,C 180,E1 -6744.551,E2 -6744.551} C_VEL
LIN {X 0,Y 481.062,Z 420.855,A -85,B 0,C 180,E1 -6745.811,E2 -6745.811} C_VEL
LIN {X 0,Y 481,Z 422.704,A -85,B 0,C 180,E1 -6746.649,E2 -6746.649} C_VEL
LIN {X 0,Y 480.943,Z 424.118,A -85,B 0,C 180,E1 -6747.487,E2 -6747.487} C_VEL
LIN {X 0,Y 480.768,Z 425.729,A -85,B 0,C 180,E1 -6749.162,E2 -6749.162} C_VEL
LIN {X 0,Y 480.759,Z 425.965,A -85,B 0,C 180,E1 -6750,E2 -6750} C_VEL
LIN {X 0,Y 480.827,Z 425.197,A -85,B 0,C 180,E1 -6751.675,E2 -6751.675} C_VEL
LIN {X 0,Y 480.943,Z 424.234,A -85,B 0,C 180,E1 -6752.513,E2 -6752.513} C_VEL
LIN {X 0,Y 480.999,Z 422.883,A -85,B 0,C 180,E1 -6753.351,E2 -6753.351} C_VEL
LIN {X 0,Y 481.035,Z 420.042,A -85,B 0,C 180,E1 -6754.609,E2 -6754.609} C_VEL
LIN {X 0,Y 481.155,Z 416.179,A -85,B 0,C 180,E1 -6755.869,E2 -6755.869} C_VEL
LIN {X 0,Y 481.345,Z 411.177,A -85,B 0,C 180,E1 -6757.129,E2 -6757.129} C_VEL
LIN {X 0,Y 481.586,Z 404.859,A -85,B 0,C 180,E1 -6758.391,E2 -6758.391} C_VEL
LIN {X 0,Y 481.917,Z 397.007,A -85,B 0,C 180,E1 -6759.655,E2 -6759.655} C_VEL
LIN {X 0,Y 482.361,Z 388.982,A -85,B 0,C 180,E1 -6760.706,E2 -6760.706} C_VEL
LIN {X 0,Y 482.735,Z 379.157,A -85,B 0,C 180,E1 -6761.761,E2 -6761.761} C_VEL
LIN {X 0,Y 483.115,Z 368.3,A -85,B 0,C 180,E1 -6762.694,E2 -6762.694} C_VEL
LIN {X 0,Y 483.542,Z 357.263,A -85,B 0,C 180,E1 -6763.447,E2 -6763.447} C_VEL
LIN {X 0,Y 483.924,Z 345.209,A -85,B 0,C 180,E1 -6764.079,E2 -6764.079} C_VEL
LIN {X 0,Y 484.021,Z 335.21,A -85,B 0,C 180,E1 -6764.479,E2 -6764.479} C_VEL
LIN {X 0,Y 481.113,Z 321.421,A -85,B 0,C 180,E1 -6764.947,E2 -6764.947} C_VEL
LIN {X 0,Y 481.064,Z 315.281,A -85,B 0,C 180,E1 -6768.267,E2 -6768.267} C_VEL
LIN {X 0,Y 481.109,Z 309.839,A -85,B 0,C 180,E1 -6771.42,E2 -6771.42} C_VEL
LIN {X 0,Y 481.17,Z 305.303,A -85,B 0,C 180,E1 -6774.14,E2 -6774.14} C_VEL
LIN {X 0,Y 481.195,Z 300.573,A -85,B 0,C 180,E1 -6777.01,E2 -6777.01} C_VEL
LIN {X 0,Y 481.24,Z 296,A -85,B 0,C 180,E1 -6779.771,E2 -6779.771} C_VEL
LIN {X 0,Y 481.324,Z 290.985,A -85,B 0,C 180,E1 -6782.701,E2 -6782.701} C_VEL
LIN {X 0,Y 481.452,Z 289.518,A -85,B 0,C 180,E1 -6783.614,E2 -6783.614} C_VEL
LIN {X 0,Y 481.61,Z 289.497,A -85,B 0,C 180,E1 -6785.712,E2 -6785.712} C_VEL
LIN {X 0,Y 481.673,Z 289.487,A -85,B 0,C 180,E1 -6788.859,E2 -6788.859} C_VEL
LIN {X 0,Y 481.655,Z 289.489,A -85,B 0,C 180,E1 -6791.913,E2 -6791.913} C_VEL
LIN {X 0,Y 481.657,Z 289.489,A -85,B 0,C 180,E1 -6794.458,E2 -6794.458} C_VEL
LIN {X 0,Y 481.65,Z 289.49,A -85,B 0,C 180,E1 -6797.839,E2 -6797.839} C_VEL
LIN {X 0,Y 481.683,Z 289.485,A -85,B 0,C 180,E1 -6800.651,E2 -6800.651} C_VEL
LIN {X 0,Y 481.62,Z 289.493,A -85,B 0,C 180,E1 -6803.378,E2 -6803.378} C_VEL
LIN {X 0,Y 481.459,Z 289.516,A -85,B 0,C 180,E1 -6806.31,E2 -6806.31} C_VEL
LIN {X 0,Y 481.363,Z 289.699,A -85,B 0,C 180,E1 -6806.804,E2 -6806.804} C_VEL
LIN {X 0,Y 481.25,Z 295.701,A -85,B 0,C 180,E1 -6810.23,E2 -6810.23} C_VEL
LIN {X 0,Y 481.208,Z 300.655,A -85,B 0,C 180,E1 -6813.079,E2 -6813.079} C_VEL
LIN {X 0,Y 481.186,Z 305.453,A -85,B 0,C 180,E1 -6815.861,E2 -6815.861} C_VEL
LIN {X 0,Y 481.162,Z 311.653,A -85,B 0,C 180,E1 -6819.479,E2 -6819.479} C_VEL
LIN {X 0,Y 481.091,Z 316.17,A -85,B 0,C 180,E1 -6822.135,E2 -6822.135} C_VEL
LIN {X 0,Y 481.132,Z 321.791,A -85,B 0,C 180,E1 -6825.311,E2 -6825.311} C_VEL
LIN {X 0,Y 483.686,Z 334.984,A -85,B 0,C 180,E1 -6825.766,E2 -6825.766} C_VEL
LIN {X 0,Y 483.467,Z 347.364,A -85,B 0,C 180,E1 -6826.283,E2 -6826.283} C_VEL
LIN {X 0,Y 483.156,Z 358.297,A -85,B 0,C 180,E1 -6826.884,E2 -6826.884} C_VEL
LIN {X 0,Y 482.833,Z 369.934,A -85,B 0,C 180,E1 -6827.709,E2 -6827.709} C_VEL
LIN {X 0,Y 482.441,Z 380.685,A -85,B 0,C 180,E1 -6828.658,E2 -6828.658} C_VEL
LIN {X 0,Y 482.043,Z 390.286,A -85,B 0,C 180,E1 -6829.712,E2 -6829.712} C_VEL
LIN {X 0,Y 481.696,Z 399.606,A -85,B 0,C 180,E1 -6830.976,E2 -6830.976} C_VEL
LIN {X 0,Y 481.398,Z 407.036,A -85,B 0,C 180,E1 -6832.239,E2 -6832.239} C_VEL
LIN {X 0,Y 481.228,Z 413.238,A -85,B 0,C 180,E1 -6833.56,E2 -6833.56} C_VEL
LIN {X 0,Y 480.965,Z 418.389,A -85,B 0,C 180,E1 -6834.97,E2 -6834.97} C_VEL
LIN {X 0,Y 481.057,Z 420.739,A -85,B 0,C 180,E1 -6835.811,E2 -6835.811} C_VEL
LIN {X 0,Y 480.999,Z 422.666,A -85,B 0,C 180,E1 -6836.649,E2 -6836.649} C_VEL
LIN {X 0,Y 480.943,Z 424.174,A -85,B 0,C 180,E1 -6837.487,E2 -6837.487} C_VEL
LIN {X 0,Y 480.771,Z 425.89,A -85,B 0,C 180,E1 -6839.162,E2 -6839.162} C_VEL
LIN {X 0,Y 480.763,Z 426.164,A -85,B 0,C 180,E1 -6840,E2 -6840} C_VEL
LIN {X 0,Y 480.772,Z 425.995,A -85,B 0,C 180,E1 -6840.838,E2 -6840.838} C_VEL
LIN {X 0,Y 480.945,Z 424.464,A -85,B 0,C 180,E1 -6842.513,E2 -6842.513} C_VEL
LIN {X 0,Y 481.025,Z 423.067,A -85,B 0,C 180,E1 -6843.35,E2 -6843.35} C_VEL
LIN {X 0,Y 481.044,Z 420.161,A -85,B 0,C 180,E1 -6844.609,E2 -6844.609} C_VEL
LIN {X 0,Y 481.151,Z 416.184,A -85,B 0,C 180,E1 -6845.869,E2 -6845.869} C_VEL
LIN {X 0,Y 481.361,Z 410.15,A -85,B 0,C 180,E1 -6847.319,E2 -6847.319} C_VEL
LIN {X 0,Y 481.615,Z 403.285,A -85,B 0,C 180,E1 -6848.602,E2 -6848.602} C_VEL
LIN {X 0,Y 481.925,Z 394.79,A -85,B 0,C 180,E1 -6849.866,E2 -6849.866} C_VEL
LIN {X 0,Y 482.229,Z 386.078,A -85,B 0,C 180,E1 -6850.921,E2 -6850.921} C_VEL
LIN {X 0,Y 482.718,Z 375.225,A -85,B 0,C 180,E1 -6851.974,E2 -6851.974} C_VEL
LIN {X 0,Y 483.003,Z 363.818,A -85,B 0,C 180,E1 -6852.865,E2 -6852.865} C_VEL
LIN {X 0,Y 483.337,Z 352.365,A -85,B 0,C 180,E1 -6853.56,E2 -6853.56} C_VEL
LIN {X 0,Y 483.703,Z 339.875,A -85,B 0,C 180,E1 -6854.139,E2 -6854.139} C_VEL
LIN {X 0,Y 483.662,Z 334.747,A -85,B 0,C 180,E1 -6854.331,E2 -6854.331} C_VEL
LIN {X 0,Y 481.23,Z 323.088,A -85,B 0,C 180,E1 -6854.754,E2 -6854.754} C_VEL
LIN {X 0,Y 481.25,Z 316.759,A -85,B 0,C 180,E1 -6858.334,E2 -6858.334} C_VEL
LIN {X 0,Y 481.247,Z 311.177,A -85,B 0,C 180,E1 -6861.413,E2 -6861.413} C_VEL
LIN {X 0,Y 481.242,Z 305.985,A -85,B 0,C 180,E1 -6864.136,E2 -6864.136} C_VEL
LIN {X 0,Y 481.205,Z 300.232,A -85,B 0,C 180,E1 -6867.012,E2 -6867.012} C_VEL
LIN {X 0,Y 481.199,Z 294.276,A -85,B 0,C 180,E1 -6869.774,E2 -6869.774} C_VEL
LIN {X 0,Y 481.208,Z 289.549,A -85,B 0,C 180,E1 -6871.822,E2 -6871.822} C_VEL
LIN {X 0,Y 481.622,Z 289.495,A -85,B 0,C 180,E1 -6874.688,E2 -6874.688} C_VEL
LIN {X 0,Y 481.656,Z 289.49,A -85,B 0,C 180,E1 -6878.007,E2 -6878.007} C_VEL
LIN {X 0,Y 481.651,Z 289.489,A -85,B 0,C 180,E1 -6881.042,E2 -6881.042} C_VEL
LIN {X 0,Y 481.661,Z 289.489,A -85,B 0,C 180,E1 -6884.457,E2 -6884.457} C_VEL
LIN {X 0,Y 481.645,Z 289.491,A -85,B 0,C 180,E1 -6887.839,E2 -6887.839} C_VEL
LIN {X 0,Y 481.707,Z 289.568,A -85,B 0,C 180,E1 -6889.078,E2 -6889.078} C_VEL
LIN {X 0,Y 483.415,Z 298.523,A -85,B 0,C 180,E1 -6892.366,E2 -6892.366} C_VEL
LIN {X 0,Y 484.11,Z 303.1,A -85,B 0,C 180,E1 -6893.988,E2 -6893.988} C_VEL
LIN {X 0,Y 483.677,Z 310.939,A -85,B 0,C 180,E1 -6896.485,E2 -6896.485} C_VEL
LIN {X 0,Y 483.268,Z 320.347,A -85,B 0,C 180,E1 -6899.403,E2 -6899.403} C_VEL
LIN {X 0,Y 482.817,Z 329.603,A -85,B 0,C 180,E1 -6902.238,E2 -6902.238} C_VEL
LIN {X 0,Y 482.507,Z 338.947,A -85,B 0,C 180,E1 -6905.014,E2 -6905.014} C_VEL
LIN {X 0,Y 482.205,Z 348.574,A -85,B 0,C 180,E1 -6907.732,E2 -6907.732} C_VEL
LIN {X 0,Y 481.877,Z 359.739,A -85,B 0,C 180,E1 -6910.843,E2 -6910.843} C_VEL
LIN {X 0,Y 481.624,Z 369.148,A -85,B 0,C 180,E1 -6913.468,E2 -6913.468} C_VEL
LIN {X 0,Y 481.431,Z 374.712,A -85,B 0,C 180,E1 -6915.036,E2 -6915.036} C_VEL
LIN {X 0,Y 483.818,Z 388.637,A -85,B 0,C 180,E1 -6915.448,E2 -6915.448} C_VEL
LIN {X 0,Y 483.793,Z 399.772,A -85,B 0,C 180,E1 -6915.863,E2 -6915.863} C_VEL
LIN {X 0,Y 483.376,Z 411.406,A -85,B 0,C 180,E1 -6916.441,E2 -6916.441} C_VEL
LIN {X 0,Y 482.899,Z 423.925,A -85,B 0,C 180,E1 -6917.265,E2 -6917.265} C_VEL
LIN {X 0,Y 482.522,Z 434.264,A -85,B 0,C 180,E1 -6918.128,E2 -6918.128} C_VEL
LIN {X 0,Y 482.081,Z 443.539,A -85,B 0,C 180,E1 -6919.075,E2 -6919.075} C_VEL
LIN {X 0,Y 481.756,Z 451.992,A -85,B 0,C 180,E1 -6920.13,E2 -6920.13} C_VEL
LIN {X 0,Y 481.426,Z 460.235,A -85,B 0,C 180,E1 -6921.394,E2 -6921.394} C_VEL
LIN {X 0,Y 481.114,Z 466.875,A -85,B 0,C 180,E1 -6922.656,E2 -6922.656} C_VEL
LIN {X 0,Y 481.022,Z 472.95,A -85,B 0,C 180,E1 -6924.13,E2 -6924.13} C_VEL
LIN {X 0,Y 480.854,Z 476.895,A -85,B 0,C 180,E1 -6925.389,E2 -6925.389} C_VEL
LIN {X 0,Y 480.891,Z 479.807,A -85,B 0,C 180,E1 -6926.649,E2 -6926.649} C_VEL
LIN {X 0,Y 480.79,Z 482.182,A -85,B 0,C 180,E1 -6928.325,E2 -6928.325} C_VEL
LIN {X 0,Y 480.743,Z 483,A -85,B 0,C 180,E1 -6930,E2 -6930} C_VEL
LIN {X 0,Y 480.79,Z 482.184,A -85,B 0,C 180,E1 -6931.675,E2 -6931.675} C_VEL
LIN {X 0,Y 480.891,Z 479.81,A -85,B 0,C 180,E1 -6933.351,E2 -6933.351} C_VEL
LIN {X 0,Y 480.854,Z 476.895,A -85,B 0,C 180,E1 -6934.611,E2 -6934.611} C_VEL
LIN {X 0,Y 481.023,Z 472.948,A -85,B 0,C 180,E1 -6935.87,E2 -6935.87} C_VEL
LIN {X 0,Y 481.116,Z 466.875,A -85,B 0,C 180,E1 -6937.344,E2 -6937.344} C_VEL
LIN {X 0,Y 481.426,Z 460.235,A -85,B 0,C 180,E1 -6938.606,E2 -6938.606} C_VEL
LIN {X 0,Y 481.756,Z 451.991,A -85,B 0,C 180,E1 -6939.87,E2 -6939.87} C_VEL
LIN {X 0,Y 482.082,Z 443.539,A -85,B 0,C 180,E1 -6940.925,E2 -6940.925} C_VEL
LIN {X 0,Y 482.582,Z 433.091,A -85,B 0,C 180,E1 -6941.978,E2 -6941.978} C_VEL
LIN {X 0,Y 482.968,Z 421.877,A -85,B 0,C 180,E1 -6942.887,E2 -6942.887} C_VEL
LIN {X 0,Y 483.345,Z 411.403,A -85,B 0,C 180,E1 -6943.56,E2 -6943.56} C_VEL
LIN {X 0,Y 483.802,Z 399.762,A -85,B 0,C 180,E1 -6944.136,E2 -6944.136} C_VEL
LIN {X 0,Y 483.88,Z 389.084,A -85,B 0,C 180,E1 -6944.537,E2 -6944.537} C_VEL
LIN {X 0,Y 481.72,Z 376.358,A -85,B 0,C 180,E1 -6944.923,E2 -6944.923} C_VEL
LIN {X 0,Y 481.431,Z 374.712,A -85,B 0,C 180,E1 -6944.964,E2 -6944.964} C_VEL
LIN {X 0,Y 481.78,Z 364.502,A -85,B 0,C 180,E1 -6947.839,E2 -6947.839} C_VEL
LIN {X 0,Y 482.077,Z 351.362,A -85,B 0,C 180,E1 -6951.375,E2 -6951.375} C_VEL
LIN {X 0,Y 482.383,Z 339.713,A -85,B 0,C 180,E1 -6954.534,E2 -6954.534} C_VEL
LIN {X 0,Y 482.666,Z 328.215,A -85,B 0,C 180,E1 -6957.772,E2 -6957.772} C_VEL
LIN {X 0,Y 483.046,Z 318.393,A -85,B 0,C 180,E1 -6960.612,E2 -6960.612} C_VEL
LIN {X 0,Y 483.464,Z 307.26,A -85,B 0,C 180,E1 -6964.045,E2 -6964.045} C_VEL
LIN {X 0,Y 483.684,Z 301.251,A -85,B 0,C 180,E1 -6966.049,E2 -6966.049} C_VEL
LIN {X 0,Y 482.812,Z 295.663,A -85,B 0,C 180,E1 -6968.182,E2 -6968.182} C_VEL
LIN {X 0,Y 481.661,Z 289.509,A -85,B 0,C 180,E1 -6970.932,E2 -6970.932} C_VEL
LIN {X 0,Y 481.656,Z 289.492,A -85,B 0,C 180,E1 -6974.458,E2 -6974.458} C_VEL
LIN {X 0,Y 481.645,Z 289.491,A -85,B 0,C 180,E1 -6977.839,E2 -6977.839} C_VEL
LIN {X 0,Y 481.663,Z 289.489,A -85,B 0,C 180,E1 -6980.654,E2 -6980.654} C_VEL
LIN {X 0,Y 481.63,Z 289.491,A -85,B 0,C 180,E1 -6983.376,E2 -6983.376} C_VEL
LIN {X 0,Y 481.712,Z 289.483,A -85,B 0,C 180,E1 -6986.33,E2 -6986.33} C_VEL
LIN {X 0,Y 481.654,Z 289.491,A -85,B 0,C 180,E1 -6989.417,E2 -6989.417} C_VEL
LIN {X 0,Y 481.697,Z 289.485,A -85,B 0,C 180,E1 -6992.168,E2 -6992.168} C_VEL
LIN {X 0,Y 481.666,Z 289.49,A -85,B 0,C 180,E1 -6994.967,E2 -6994.967} C_VEL
LIN {X 0,Y 481.569,Z 289.636,A -85,B 0,C 180,E1 -6995.881,E2 -6995.881} C_VEL
LIN {X 0,Y 481.588,Z 292.319,A -85,B 0,C 180,E1 -6999.064,E2 -6999.064} C_VEL
LIN {X 0,Y 481.479,Z 295.019,A -85,B 0,C 180,E1 -7002.15,E2 -7002.15} C_VEL
LIN {X 0,Y 481.464,Z 298.045,A -85,B 0,C 180,E1 -7005.382,E2 -7005.382} C_VEL
LIN {X 0,Y 483.957,Z 307.95,A -85,B 0,C 180,E1 -7005.761,E2 -7005.761} C_VEL
LIN {X 0,Y 483.681,Z 320.633,A -85,B 0,C 180,E1 -7006.289,E2 -7006.289} C_VEL
LIN {X 0,Y 483.409,Z 332.071,A -85,B 0,C 180,E1 -7006.926,E2 -7006.926} C_VEL
LIN {X 0,Y 483.062,Z 343.175,A -85,B 0,C 180,E1 -7007.715,E2 -7007.715} C_VEL
LIN {X 0,Y 482.708,Z 353.764,A -85,B 0,C 180,E1 -7008.664,E2 -7008.664} C_VEL
LIN {X 0,Y 482.345,Z 363.307,A -85,B 0,C 180,E1 -7009.718,E2 -7009.718} C_VEL
LIN {X 0,Y 482.068,Z 371.115,A -85,B 0,C 180,E1 -7010.772,E2 -7010.772} C_VEL
LIN {X 0,Y 481.739,Z 378.698,A -85,B 0,C 180,E1 -7012.034,E2 -7012.034} C_VEL
LIN {X 0,Y 481.462,Z 384.747,A -85,B 0,C 180,E1 -7013.294,E2 -7013.294} C_VEL
LIN {X 0,Y 481.306,Z 389.505,A -85,B 0,C 180,E1 -7014.554,E2 -7014.554} C_VEL
LIN {X 0,Y 481.267,Z 393.124,A -85,B 0,C 180,E1 -7015.813,E2 -7015.813} C_VEL
LIN {X 0,Y 481.12,Z 394.985,A -85,B 0,C 180,E1 -7016.65,E2 -7016.65} C_VEL
LIN {X 0,Y 480.994,Z 396.404,A -85,B 0,C 180,E1 -7017.488,E2 -7017.488} C_VEL
LIN {X 0,Y 480.9,Z 397.957,A -85,B 0,C 180,E1 -7019.163,E2 -7019.163} C_VEL
LIN {X 0,Y 480.89,Z 398.149,A -85,B 0,C 180,E1 -7020,E2 -7020} C_VEL
LIN {X 0,Y 480.892,Z 397.916,A -85,B 0,C 180,E1 -7020.837,E2 -7020.837} C_VEL
LIN {X 0,Y 480.971,Z 396.238,A -85,B 0,C 180,E1 -7022.512,E2 -7022.512} C_VEL
LIN {X 0,Y 481.114,Z 394.795,A -85,B 0,C 180,E1 -7023.35,E2 -7023.35} C_VEL
LIN {X 0,Y 481.245,Z 391.799,A -85,B 0,C 180,E1 -7024.607,E2 -7024.607} C_VEL
LIN {X 0,Y 481.225,Z 387.771,A -85,B 0,C 180,E1 -7025.868,E2 -7025.868} C_VEL
LIN {X 0,Y 481.481,Z 381.893,A -85,B 0,C 180,E1 -7027.265,E2 -7027.265} C_VEL
LIN {X 0,Y 481.741,Z 374.745,A -85,B 0,C 180,E1 -7028.6,E2 -7028.6} C_VEL
LIN {X 0,Y 482.027,Z 366.294,A -85,B 0,C 180,E1 -7029.864,E2 -7029.864} C_VEL
LIN {X 0,Y 482.413,Z 357.569,A -85,B 0,C 180,E1 -7030.917,E2 -7030.917} C_VEL
LIN {X 0,Y 482.8,Z 346.839,A -85,B 0,C 180,E1 -7031.972,E2 -7031.972} C_VEL
LIN {X 0,Y 483.166,Z 335.373,A -85,B 0,C 180,E1 -7032.871,E2 -7032.871} C_VEL
LIN {X 0,Y 483.479,Z 324.276,A -85,B 0,C 180,E1 -7033.556,E2 -7033.556} C_VEL
LIN {X 0,Y 483.836,Z 310.764,A -85,B 0,C 180,E1 -7034.189,E2 -7034.189} C_VEL
LIN {X 0,Y 483.59,Z 305.668,A -85,B 0,C 180,E1 -7034.384,E2 -7034.384} C_VEL
LIN {X 0,Y 481.093,Z 294.867,A -85,B 0,C 180,E1 -7034.771,E2 -7034.771} C_VEL
LIN {X 0,Y 481.05,Z 290.828,A -85,B 0,C 180,E1 -7038.262,E2 -7038.262} C_VEL
LIN {X 0,Y 481.066,Z 289.565,A -85,B 0,C 180,E1 -7039.634,E2 -7039.634} C_VEL
LIN {X 0,Y 481.353,Z 289.528,A -85,B 0,C 180,E1 -7042.31,E2 -7042.31} C_VEL
LIN {X 0,Y 481.663,Z 289.483,A -85,B 0,C 180,E1 -7045.223,E2 -7045.223} C_VEL
LIN {X 0,Y 481.696,Z 289.478,A -85,B 0,C 180,E1 -7047.832,E2 -7047.832} C_VEL
LIN {X 0,Y 481.647,Z 289.487,A -85,B 0,C 180,E1 -7050.711,E2 -7050.711} C_VEL
LIN {X 0,Y 481.7,Z 289.48,A -85,B 0,C 180,E1 -7053.733,E2 -7053.733} C_VEL
LIN {X 0,Y 481.629,Z 289.491,A -85,B 0,C 180,E1 -7056.747,E2 -7056.747} C_VEL
LIN {X 0,Y 481.68,Z 289.487,A -85,B 0,C 180,E1 -7059.94,E2 -7059.94} C_VEL
LIN {X 0,Y 481.642,Z 289.488,A -85,B 0,C 180,E1 -7063.3,E2 -7063.3} C_VEL
LIN {X 0,Y 481.661,Z 289.488,A -85,B 0,C 180,E1 -7065.641,E2 -7065.641} C_VEL
LIN {X 0,Y 481.659,Z 289.484,A -85,B 0,C 180,E1 -7068.958,E2 -7068.958} C_VEL
LIN {X 0,Y 481.657,Z 289.488,A -85,B 0,C 180,E1 -7071.993,E2 -7071.993} C_VEL
LIN {X 0,Y 481.596,Z 289.495,A -85,B 0,C 180,E1 -7074.807,E2 -7074.807} C_VEL
LIN {X 0,Y 481.424,Z 289.616,A -85,B 0,C 180,E1 -7076.621,E2 -7076.621} C_VEL
LIN {X 0,Y 481.268,Z 294.598,A -85,B 0,C 180,E1 -7079.495,E2 -7079.495} C_VEL
LIN {X 0,Y 481.208,Z 298.993,A -85,B 0,C 180,E1 -7082.137,E2 -7082.137} C_VEL
LIN {X 0,Y 481.171,Z 301.878,A -85,B 0,C 180,E1 -7083.879,E2 -7083.879} C_VEL
LIN {X 0,Y 480.522,Z 303.077,A -85,B 0,C 180,E1 -7084.562,E2 -7084.562} C_VEL
LIN {X 0,Y 477.663,Z 305.196,A -85,B 0,C 180,E1 -7085.668,E2 -7085.668} C_VEL
LIN {X 0,Y 475.221,Z 306.91,A -85,B 0,C 180,E1 -7086.558,E2 -7086.558} C_VEL
LIN {X 0,Y 474.154,Z 308.157,A -85,B 0,C 180,E1 -7087.248,E2 -7087.248} C_VEL
LIN {X 0,Y 474.058,Z 308.556,A -85,B 0,C 180,E1 -7087.483,E2 -7087.483} C_VEL
LIN {X 0,Y 474.01,Z 312.929,A -85,B 0,C 180,E1 -7090.061,E2 -7090.061} C_VEL
LIN {X 0,Y 473.968,Z 317.706,A -85,B 0,C 180,E1 -7092.749,E2 -7092.749} C_VEL
LIN {X 0,Y 474.067,Z 321.913,A -85,B 0,C 180,E1 -7094.923,E2 -7094.923} C_VEL
LIN {X 0,Y 476.997,Z 335.289,A -85,B 0,C 180,E1 -7095.385,E2 -7095.385} C_VEL
LIN {X 0,Y 477.176,Z 341.052,A -85,B 0,C 180,E1 -7095.609,E2 -7095.609} C_VEL
LIN {X 0,Y 476.834,Z 352.387,A -85,B 0,C 180,E1 -7096.143,E2 -7096.143} C_VEL
LIN {X 0,Y 476.409,Z 364.051,A -85,B 0,C 180,E1 -7096.867,E2 -7096.867} C_VEL
LIN {X 0,Y 475.983,Z 375.148,A -85,B 0,C 180,E1 -7097.746,E2 -7097.746} C_VEL
LIN {X 0,Y 475.58,Z 384.891,A -85,B 0,C 180,E1 -7098.708,E2 -7098.708} C_VEL
LIN {X 0,Y 475.12,Z 393.713,A -85,B 0,C 180,E1 -7099.775,E2 -7099.775} C_VEL
LIN {X 0,Y 474.717,Z 402.317,A -85,B 0,C 180,E1 -7101.057,E2 -7101.057} C_VEL
LIN {X 0,Y 474.401,Z 409.216,A -85,B 0,C 180,E1 -7102.338,E2 -7102.338} C_VEL
LIN {X 0,Y 474.178,Z 415.257,A -85,B 0,C 180,E1 -7103.77,E2 -7103.77} C_VEL
LIN {X 0,Y 473.992,Z 420.211,A -85,B 0,C 180,E1 -7105.322,E2 -7105.322} C_VEL
LIN {X 0,Y 473.927,Z 423.119,A -85,B 0,C 180,E1 -7106.599,E2 -7106.599} C_VEL
LIN {X 0,Y 473.885,Z 424.531,A -85,B 0,C 180,E1 -7107.45,E2 -7107.45} C_VEL
LIN {X 0,Y 473.696,Z 426.143,A -85,B 0,C 180,E1 -7109.15,E2 -7109.15} C_VEL
LIN {X 0,Y 473.685,Z 426.379,A -85,B 0,C 180,E1 -7110,E2 -7110} C_VEL
LIN {X 0,Y 473.762,Z 425.61,A -85,B 0,C 180,E1 -7111.7,E2 -7111.7} C_VEL
LIN {X 0,Y 473.885,Z 424.646,A -85,B 0,C 180,E1 -7112.55,E2 -7112.55} C_VEL
LIN {X 0,Y 473.926,Z 423.296,A -85,B 0,C 180,E1 -7113.401,E2 -7113.401} C_VEL
LIN {X 0,Y 473.973,Z 420.454,A -85,B 0,C 180,E1 -7114.678,E2 -7114.678} C_VEL
LIN {X 0,Y 474.183,Z 415.583,A -85,B 0,C 180,E1 -7116.231,E2 -7116.231} C_VEL
LIN {X 0,Y 474.383,Z 409.626,A -85,B 0,C 180,E1 -7117.662,E2 -7117.662} C_VEL
LIN {X 0,Y 474.702,Z 402.86,A -85,B 0,C 180,E1 -7118.943,E2 -7118.943} C_VEL
LIN {X 0,Y 475.068,Z 394.382,A -85,B 0,C 180,E1 -7120.226,E2 -7120.226} C_VEL
LIN {X 0,Y 475.53,Z 385.694,A -85,B 0,C 180,E1 -7121.293,E2 -7121.293} C_VEL
LIN {X 0,Y 475.943,Z 376.159,A -85,B 0,C 180,E1 -7122.255,E2 -7122.255} C_VEL
LIN {X 0,Y 476.337,Z 364.788,A -85,B 0,C 180,E1 -7123.173,E2 -7123.173} C_VEL
LIN {X 0,Y 476.807,Z 353.968,A -85,B 0,C 180,E1 -7123.858,E2 -7123.858} C_VEL
LIN {X 0,Y 477.137,Z 341.918,A -85,B 0,C 180,E1 -7124.447,E2 -7124.447} C_VEL
LIN {X 0,Y 477.107,Z 335.967,A -85,B 0,C 180,E1 -7124.679,E2 -7124.679} C_VEL
LIN {X 0,Y 474.36,Z 323.256,A -85,B 0,C 180,E1 -7125.13,E2 -7125.13} C_VEL
LIN {X 0,Y 474.072,Z 321.698,A -85,B 0,C 180,E1 -7125.202,E2 -7125.202} C_VEL
LIN {X 0,Y 474.015,Z 315.798,A -85,B 0,C 180,E1 -7128.395,E2 -7128.395} C_VEL
LIN {X 0,Y 474.052,Z 310.007,A -85,B 0,C 180,E1 -7131.755,E2 -7131.755} C_VEL
LIN {X 0,Y 474.109,Z 305.419,A -85,B 0,C 180,E1 -7134.523,E2 -7134.523} C_VEL
LIN {X 0,Y 474.142,Z 300.753,A -85,B 0,C 180,E1 -7137.355,E2 -7137.355} C_VEL
LIN {X 0,Y 474.191,Z 295.949,A -85,B 0,C 180,E1 -7140.26,E2 -7140.26} C_VEL
LIN {X 0,Y 474.398,Z 290.397,A -85,B 0,C 180,E1 -7143.592,E2 -7143.592} C_VEL
LIN {X 0,Y 474.579,Z 290.371,A -85,B 0,C 180,E1 -7146.325,E2 -7146.325} C_VEL
LIN {X 0,Y 474.631,Z 290.366,A -85,B 0,C 180,E1 -7149.648,E2 -7149.648} C_VEL
LIN {X 0,Y 474.617,Z 290.367,A -85,B 0,C 180,E1 -7152.934,E2 -7152.934} C_VEL
LIN {X 0,Y 474.608,Z 290.367,A -85,B 0,C 180,E1 -7155.895,E2 -7155.895} C_VEL
LIN {X 0,Y 474.63,Z 290.365,A -85,B 0,C 180,E1 -7159.041,E2 -7159.041} C_VEL
LIN {X 0,Y 474.611,Z 290.366,A -85,B 0,C 180,E1 -7161.704,E2 -7161.704} C_VEL
LIN {X 0,Y 474.554,Z 290.371,A -85,B 0,C 180,E1 -7164.719,E2 -7164.719} C_VEL
LIN {X 0,Y 474.312,Z 290.612,A -85,B 0,C 180,E1 -7166.874,E2 -7166.874} C_VEL
LIN {X 0,Y 474.195,Z 295.621,A -85,B 0,C 180,E1 -7169.741,E2 -7169.741} C_VEL
LIN {X 0,Y 474.149,Z 300.904,A -85,B 0,C 180,E1 -7172.791,E2 -7172.791} C_VEL
LIN {X 0,Y 474.117,Z 305.504,A -85,B 0,C 180,E1 -7175.477,E2 -7175.477} C_VEL
LIN {X 0,Y 474.082,Z 310.267,A -85,B 0,C 180,E1 -7178.247,E2 -7178.247} C_VEL
LIN {X 0,Y 474.037,Z 314.897,A -85,B 0,C 180,E1 -7180.963,E2 -7180.963} C_VEL
LIN {X 0,Y 474.055,Z 320.995,A -85,B 0,C 180,E1 -7184.523,E2 -7184.523} C_VEL
LIN {X 0,Y 474.081,Z 321.991,A -85,B 0,C 180,E1 -7185.101,E2 -7185.101} C_VEL
LIN {X 0,Y 476.781,Z 335.809,A -85,B 0,C 180,E1 -7185.597,E2 -7185.597} C_VEL
LIN {X 0,Y 476.539,Z 348.326,A -85,B 0,C 180,E1 -7186.134,E2 -7186.134} C_VEL
LIN {X 0,Y 476.173,Z 359.588,A -85,B 0,C 180,E1 -7186.776,E2 -7186.776} C_VEL
LIN {X 0,Y 475.861,Z 371.319,A -85,B 0,C 180,E1 -7187.634,E2 -7187.634} C_VEL
LIN {X 0,Y 475.446,Z 381.869,A -85,B 0,C 180,E1 -7188.597,E2 -7188.597} C_VEL
LIN {X 0,Y 475.062,Z 390.477,A -85,B 0,C 180,E1 -7189.559,E2 -7189.559} C_VEL
LIN {X 0,Y 474.683,Z 399.847,A -85,B 0,C 180,E1 -7190.842,E2 -7190.842} C_VEL
LIN {X 0,Y 474.368,Z 407.329,A -85,B 0,C 180,E1 -7192.123,E2 -7192.123} C_VEL
LIN {X 0,Y 474.182,Z 413.848,A -85,B 0,C 180,E1 -7193.532,E2 -7193.532} C_VEL
LIN {X 0,Y 473.898,Z 418.757,A -85,B 0,C 180,E1 -7194.895,E2 -7194.895} C_VEL
LIN {X 0,Y 473.999,Z 421.124,A -85,B 0,C 180,E1 -7195.748,E2 -7195.748} C_VEL
LIN {X 0,Y 473.927,Z 423.064,A -85,B 0,C 180,E1 -7196.599,E2 -7196.599} C_VEL
LIN {X 0,Y 473.885,Z 424.589,A -85,B 0,C 180,E1 -7197.45,E2 -7197.45} C_VEL
LIN {X 0,Y 473.699,Z 426.324,A -85,B 0,C 180,E1 -7199.15,E2 -7199.15} C_VEL
LIN {X 0,Y 473.689,Z 426.607,A -85,B 0,C 180,E1 -7200,E2 -7200} C_VEL
LIN {X 0,Y 473.7,Z 426.443,A -85,B 0,C 180,E1 -7200.85,E2 -7200.85} C_VEL
LIN {X 0,Y 473.888,Z 424.915,A -85,B 0,C 180,E1 -7202.55,E2 -7202.55} C_VEL
LIN {X 0,Y 473.95,Z 423.516,A -85,B 0,C 180,E1 -7203.4,E2 -7203.4} C_VEL
LIN {X 0,Y 473.983,Z 420.602,A -85,B 0,C 180,E1 -7204.678,E2 -7204.678} C_VEL
LIN {X 0,Y 474.11,Z 416.612,A -85,B 0,C 180,E1 -7205.956,E2 -7205.956} C_VEL
LIN {X 0,Y 474.339,Z 410.459,A -85,B 0,C 180,E1 -7207.449,E2 -7207.449} C_VEL
LIN {X 0,Y 474.59,Z 403.659,A -85,B 0,C 180,E1 -7208.731,E2 -7208.731} C_VEL
LIN {X 0,Y 474.943,Z 395.157,A -85,B 0,C 180,E1 -7210.013,E2 -7210.013} C_VEL
LIN {X 0,Y 475.273,Z 386.431,A -85,B 0,C 180,E1 -7211.083,E2 -7211.083} C_VEL
LIN {X 0,Y 475.785,Z 375.569,A -85,B 0,C 180,E1 -7212.151,E2 -7212.151} C_VEL
LIN {X 0,Y 476.068,Z 364.79,A -85,B 0,C 180,E1 -7213.009,E2 -7213.009} C_VEL
LIN {X 0,Y 476.447,Z 352.618,A -85,B 0,C 180,E1 -7213.76,E2 -7213.76} C_VEL
LIN {X 0,Y 476.827,Z 340.074,A -85,B 0,C 180,E1 -7214.347,E2 -7214.347} C_VEL
LIN {X 0,Y 476.65,Z 335.011,A -85,B 0,C 180,E1 -7214.544,E2 -7214.544} C_VEL
LIN {X 0,Y 474.199,Z 323.59,A -85,B 0,C 180,E1 -7214.977,E2 -7214.977} C_VEL
LIN {X 0,Y 474.196,Z 317.439,A -85,B 0,C 180,E1 -7218.461,E2 -7218.461} C_VEL
LIN {X 0,Y 474.21,Z 311.439,A -85,B 0,C 180,E1 -7221.747,E2 -7221.747} C_VEL
LIN {X 0,Y 474.178,Z 306.15,A -85,B 0,C 180,E1 -7224.519,E2 -7224.519} C_VEL
LIN {X 0,Y 474.148,Z 300.454,A -85,B 0,C 180,E1 -7227.355,E2 -7227.355} C_VEL
LIN {X 0,Y 474.159,Z 294.193,A -85,B 0,C 180,E1 -7230.262,E2 -7230.262} C_VEL
LIN {X 0,Y 474.18,Z 290.424,A -85,B 0,C 180,E1 -7231.871,E2 -7231.871} C_VEL
LIN {X 0,Y 474.543,Z 290.377,A -85,B 0,C 180,E1 -7234.248,E2 -7234.248} C_VEL
LIN {X 0,Y 474.573,Z 290.372,A -85,B 0,C 180,E1 -7236.899,E2 -7236.899} C_VEL
LIN {X 0,Y 474.615,Z 290.366,A -85,B 0,C 180,E1 -7239.645,E2 -7239.645} C_VEL
LIN {X 0,Y 474.602,Z 290.367,A -85,B 0,C 180,E1 -7242.233,E2 -7242.233} C_VEL
LIN {X 0,Y 474.623,Z 290.365,A -85,B 0,C 180,E1 -7245.297,E2 -7245.297} C_VEL
LIN {X 0,Y 474.674,Z 290.551,A -85,B 0,C 180,E1 -7248.779,E2 -7248.779} C_VEL
LIN {X 0,Y 476.185,Z 298.318,A -85,B 0,C 180,E1 -7251.693,E2 -7251.693} C_VEL
LIN {X 0,Y 477.184,Z 304.513,A -85,B 0,C 180,E1 -7253.905,E2 -7253.905} C_VEL
LIN {X 0,Y 476.714,Z 312.278,A -85,B 0,C 180,E1 -7256.437,E2 -7256.437} C_VEL
LIN {X 0,Y 476.28,Z 321.625,A -85,B 0,C 180,E1 -7259.397,E2 -7259.397} C_VEL
LIN {X 0,Y 475.749,Z 332.418,A -85,B 0,C 180,E1 -7262.745,E2 -7262.745} C_VEL
LIN {X 0,Y 475.397,Z 343.412,A -85,B 0,C 180,E1 -7266.012,E2 -7266.012} C_VEL
LIN {X 0,Y 475.007,Z 354.61,A -85,B 0,C 180,E1 -7269.201,E2 -7269.201} C_VEL
LIN {X 0,Y 474.677,Z 365.741,A -85,B 0,C 180,E1 -7272.331,E2 -7272.331} C_VEL
LIN {X 0,Y 474.389,Z 374.634,A -85,B 0,C 180,E1 -7274.809,E2 -7274.809} C_VEL
LIN {X 0,Y 476.788,Z 388.636,A -85,B 0,C 180,E1 -7275.229,E2 -7275.229} C_VEL
LIN {X 0,Y 477.065,Z 392.976,A -85,B 0,C 180,E1 -7275.387,E2 -7275.387} C_VEL
LIN {X 0,Y 476.722,Z 405.487,A -85,B 0,C 180,E1 -7275.922,E2 -7275.922} C_VEL
LIN {X 0,Y 476.286,Z 416.937,A -85,B 0,C 180,E1 -7276.583,E2 -7276.583} C_VEL
LIN {X 0,Y 475.836,Z 428.208,A -85,B 0,C 180,E1 -7277.418,E2 -7277.418} C_VEL
LIN {X 0,Y 475.414,Z 438.603,A -85,B 0,C 180,E1 -7278.38,E2 -7278.38} C_VEL
LIN {X 0,Y 474.932,Z 447.112,A -85,B 0,C 180,E1 -7279.34,E2 -7279.34} C_VEL
LIN {X 0,Y 474.604,Z 454.96,A -85,B 0,C 180,E1 -7280.41,E2 -7280.41} C_VEL
LIN {X 0,Y 474.266,Z 462.622,A -85,B 0,C 180,E1 -7281.693,E2 -7281.693} C_VEL
LIN {X 0,Y 473.982,Z 469.679,A -85,B 0,C 180,E1 -7283.187,E2 -7283.187} C_VEL
LIN {X 0,Y 473.915,Z 474.372,A -85,B 0,C 180,E1 -7284.468,E2 -7284.468} C_VEL
LIN {X 0,Y 473.752,Z 477.957,A -85,B 0,C 180,E1 -7285.746,E2 -7285.746} C_VEL
LIN {X 0,Y 473.799,Z 479.807,A -85,B 0,C 180,E1 -7286.598,E2 -7286.598} C_VEL
LIN {X 0,Y 473.695,Z 482.182,A -85,B 0,C 180,E1 -7288.3,E2 -7288.3} C_VEL
LIN {X 0,Y 473.688,Z 482.785,A -85,B 0,C 180,E1 -7289.15,E2 -7289.15} C_VEL
LIN {X 0,Y 473.669,Z 483,A -85,B 0,C 180,E1 -7290,E2 -7290} C_VEL
LIN {X 0,Y 473.688,Z 482.786,A -85,B 0,C 180,E1 -7290.85,E2 -7290.85} C_VEL
LIN {X 0,Y 473.724,Z 481.196,A -85,B 0,C 180,E1 -7292.551,E2 -7292.551} C_VEL
LIN {X 0,Y 473.799,Z 479.81,A -85,B 0,C 180,E1 -7293.402,E2 -7293.402} C_VEL
LIN {X 0,Y 473.776,Z 476.895,A -85,B 0,C 180,E1 -7294.68,E2 -7294.68} C_VEL
LIN {X 0,Y 473.942,Z 472.948,A -85,B 0,C 180,E1 -7295.958,E2 -7295.958} C_VEL
LIN {X 0,Y 474.049,Z 466.875,A -85,B 0,C 180,E1 -7297.454,E2 -7297.454} C_VEL
LIN {X 0,Y 474.377,Z 460.235,A -85,B 0,C 180,E1 -7298.735,E2 -7298.735} C_VEL
LIN {X 0,Y 474.751,Z 451.992,A -85,B 0,C 180,E1 -7300.017,E2 -7300.017} C_VEL
LIN {X 0,Y 475.101,Z 443.539,A -85,B 0,C 180,E1 -7301.087,E2 -7301.087} C_VEL
LIN {X 0,Y 475.621,Z 433.111,A -85,B 0,C 180,E1 -7302.154,E2 -7302.154} C_VEL
LIN {X 0,Y 476.028,Z 422.039,A -85,B 0,C 180,E1 -7303.066,E2 -7303.066} C_VEL
LIN {X 0,Y 476.43,Z 411.402,A -85,B 0,C 180,E1 -7303.761,E2 -7303.761} C_VEL
LIN {X 0,Y 476.9,Z 399.762,A -85,B 0,C 180,E1 -7304.345,E2 -7304.345} C_VEL
LIN {X 0,Y 477.021,Z 390.301,A -85,B 0,C 180,E1 -7304.709,E2 -7304.709} C_VEL
LIN {X 0,Y 474.866,Z 377.426,A -85,B 0,C 180,E1 -7305.122,E2 -7305.122} C_VEL
LIN {X 0,Y 474.389,Z 374.608,A -85,B 0,C 180,E1 -7305.191,E2 -7305.191} C_VEL
LIN {X 0,Y 474.706,Z 363.844,A -85,B 0,C 180,E1 -7308.114,E2 -7308.114} C_VEL
LIN {X 0,Y 474.974,Z 352.457,A -85,B 0,C 180,E1 -7311.222,E2 -7311.222} C_VEL
LIN {X 0,Y 475.305,Z 340.724,A -85,B 0,C 180,E1 -7314.457,E2 -7314.457} C_VEL
LIN {X 0,Y 475.606,Z 329.91,A -85,B 0,C 180,E1 -7317.549,E2 -7317.549} C_VEL
LIN {X 0,Y 476.035,Z 319.515,A -85,B 0,C 180,E1 -7320.613,E2 -7320.613} C_VEL
LIN {X 0,Y 476.549,Z 307.803,A -85,B 0,C 180,E1 -7324.323,E2 -7324.323} C_VEL
LIN {X 0,Y 476.727,Z 302.555,A -85,B 0,C 180,E1 -7326.135,E2 -7326.135} C_VEL
LIN {X 0,Y 475.79,Z 296.632,A -85,B 0,C 180,E1 -7328.475,E2 -7328.475} C_VEL
LIN {X 0,Y 474.62,Z 290.471,A -85,B 0,C 180,E1 -7331.391,E2 -7331.391} C_VEL
LIN {X 0,Y 474.618,Z 290.368,A -85,B 0,C 180,E1 -7334.702,E2 -7334.702} C_VEL
LIN {X 0,Y 474.617,Z 290.368,A -85,B 0,C 180,E1 -7338.214,E2 -7338.214} C_VEL
LIN {X 0,Y 474.614,Z 290.366,A -85,B 0,C 180,E1 -7341.543,E2 -7341.543} C_VEL
LIN {X 0,Y 474.627,Z 290.364,A -85,B 0,C 180,E1 -7344.726,E2 -7344.726} C_VEL
LIN {X 0,Y 474.638,Z 290.365,A -85,B 0,C 180,E1 -7347.788,E2 -7347.788} C_VEL
LIN {X 0,Y 474.627,Z 290.365,A -85,B 0,C 180,E1 -7350.885,E2 -7350.885} C_VEL
LIN {X 0,Y 474.629,Z 290.367,A -85,B 0,C 180,E1 -7353.626,E2 -7353.626} C_VEL
LIN {X 0,Y 474.582,Z 290.502,A -85,B 0,C 180,E1 -7355.503,E2 -7355.503} C_VEL
LIN {X 0,Y 474.595,Z 293.316,A -85,B 0,C 180,E1 -7358.897,E2 -7358.897} C_VEL
LIN {X 0,Y 474.5,Z 295.87,A -85,B 0,C 180,E1 -7361.878,E2 -7361.878} C_VEL
LIN {X 0,Y 474.405,Z 298.768,A -85,B 0,C 180,E1 -7365.153,E2 -7365.153} C_VEL
LIN {X 0,Y 477.075,Z 309.252,A -85,B 0,C 180,E1 -7365.578,E2 -7365.578} C_VEL
LIN {X 0,Y 476.836,Z 322.306,A -85,B 0,C 180,E1 -7366.143,E2 -7366.143} C_VEL
LIN {X 0,Y 476.506,Z 334.185,A -85,B 0,C 180,E1 -7366.829,E2 -7366.829} C_VEL
LIN {X 0,Y 476.141,Z 345.107,A -85,B 0,C 180,E1 -7367.642,E2 -7367.642} C_VEL
LIN {X 0,Y 475.767,Z 355.501,A -85,B 0,C 180,E1 -7368.605,E2 -7368.605} C_VEL
LIN {X 0,Y 475.407,Z 363.999,A -85,B 0,C 180,E1 -7369.567,E2 -7369.567} C_VEL
LIN {X 0,Y 475.113,Z 371.802,A -85,B 0,C 180,E1 -7370.635,E2 -7370.635} C_VEL
LIN {X 0,Y 474.764,Z 379.388,A -85,B 0,C 180,E1 -7371.916,E2 -7371.916} C_VEL
LIN {X 0,Y 474.458,Z 385.436,A -85,B 0,C 180,E1 -7373.194,E2 -7373.194} C_VEL
LIN {X 0,Y 474.282,Z 390.203,A -85,B 0,C 180,E1 -7374.473,E2 -7374.473} C_VEL
LIN {X 0,Y 474.235,Z 393.826,A -85,B 0,C 180,E1 -7375.751,E2 -7375.751} C_VEL
LIN {X 0,Y 474.077,Z 395.688,A -85,B 0,C 180,E1 -7376.6,E2 -7376.6} C_VEL
LIN {X 0,Y 473.936,Z 397.108,A -85,B 0,C 180,E1 -7377.45,E2 -7377.45} C_VEL
LIN {X 0,Y 473.835,Z 398.651,A -85,B 0,C 180,E1 -7379.15,E2 -7379.15} C_VEL
LIN {X 0,Y 473.824,Z 398.836,A -85,B 0,C 180,E1 -7380,E2 -7380} C_VEL
LIN {X 0,Y 473.826,Z 398.594,A -85,B 0,C 180,E1 -7380.85,E2 -7380.85} C_VEL
LIN {X 0,Y 473.915,Z 396.89,A -85,B 0,C 180,E1 -7382.55,E2 -7382.55} C_VEL
LIN {X 0,Y 474.071,Z 395.43,A -85,B 0,C 180,E1 -7383.4,E2 -7383.4} C_VEL
LIN {X 0,Y 474.199,Z 392.409,A -85,B 0,C 180,E1 -7384.676,E2 -7384.676} C_VEL
LIN {X 0,Y 474.183,Z 388.35,A -85,B 0,C 180,E1 -7385.955,E2 -7385.955} C_VEL
LIN {X 0,Y 474.472,Z 382.531,A -85,B 0,C 180,E1 -7387.351,E2 -7387.351} C_VEL
LIN {X 0,Y 474.735,Z 375.236,A -85,B 0,C 180,E1 -7388.728,E2 -7388.728} C_VEL
LIN {X 0,Y 475.059,Z 366.722,A -85,B 0,C 180,E1 -7390.011,E2 -7390.011} C_VEL
LIN {X 0,Y 475.444,Z 357.946,A -85,B 0,C 180,E1 -7391.079,E2 -7391.079} C_VEL
LIN {X 0,Y 475.879,Z 347.152,A -85,B 0,C 180,E1 -7392.149,E2 -7392.149} C_VEL
LIN {X 0,Y 476.234,Z 336.207,A -85,B 0,C 180,E1 -7393.019,E2 -7393.019} C_VEL
LIN {X 0,Y 476.585,Z 324.4,A -85,B 0,C 180,E1 -7393.756,E2 -7393.756} C_VEL
LIN {X 0,Y 476.929,Z 312.05,A -85,B 0,C 180,E1 -7394.344,E2 -7394.344} C_VEL
LIN {X 0,Y 476.743,Z 306.948,A -85,B 0,C 180,E1 -7394.546,E2 -7394.546} C_VEL
LIN {X 0,Y 474.046,Z 295.366,A -85,B 0,C 180,E1 -7394.982,E2 -7394.982} C_VEL
LIN {X 0,Y 474.003,Z 291.42,A -85,B 0,C 180,E1 -7398.391,E2 -7398.391} C_VEL
LIN {X 0,Y 473.972,Z 290.667,A -85,B 0,C 180,E1 -7399.039,E2 -7399.039} C_VEL
LIN {X 0,Y 474.252,Z 290.411,A -85,B 0,C 180,E1 -7401.745,E2 -7401.745} C_VEL
LIN {X 0,Y 474.548,Z 290.376,A -85,B 0,C 180,E1 -7404.499,E2 -7404.499} C_VEL
LIN {X 0,Y 474.676,Z 290.353,A -85,B 0,C 180,E1 -7407.332,E2 -7407.332} C_VEL
LIN {X 0,Y 474.608,Z 290.366,A -85,B 0,C 180,E1 -7410.23,E2 -7410.23} C_VEL
LIN {X 0,Y 474.646,Z 290.358,A -85,B 0,C 180,E1 -7413.22,E2 -7413.22} C_VEL
LIN {X 0,Y 474.592,Z 290.371,A -85,B 0,C 180,E1 -7416.323,E2 -7416.323} C_VEL
LIN {X 0,Y 474.63,Z 290.362,A -85,B 0,C 180,E1 -7419.648,E2 -7419.648} C_VEL
LIN {X 0,Y 474.618,Z 290.362,A -85,B 0,C 180,E1 -7422.934,E2 -7422.934} C_VEL
LIN {X 0,Y 474.613,Z 290.369,A -85,B 0,C 180,E1 -7425.895,E2 -7425.895} C_VEL
LIN {X 0,Y 474.63,Z 290.36,A -85,B 0,C 180,E1 -7429.041,E2 -7429.041} C_VEL
LIN {X 0,Y 474.613,Z 290.368,A -85,B 0,C 180,E1 -7431.704,E2 -7431.704} C_VEL
LIN {X 0,Y 474.569,Z 290.371,A -85,B 0,C 180,E1 -7434.721,E2 -7434.721} C_VEL
LIN {X 0,Y 474.364,Z 290.452,A -85,B 0,C 180,E1 -7436.64,E2 -7436.64} C_VEL
LIN {X 0,Y 474.186,Z 295.778,A -85,B 0,C 180,E1 -7439.74,E2 -7439.74} C_VEL
LIN {X 0,Y 474.144,Z 300.836,A -85,B 0,C 180,E1 -7442.792,E2 -7442.792} C_VEL
LIN {X 0,Y 474.108,Z 305.243,A -85,B 0,C 180,E1 -7445.477,E2 -7445.477} C_VEL
LIN {X 0,Y 474.058,Z 308.556,A -85,B 0,C 180,E1 -7447.483,E2 -7447.483} C_VEL
LIN {X 0,Y 473.364,Z 309.796,A -85,B 0,C 180,E1 -7448.176,E2 -7448.176} C_VEL
LIN {X 0,Y 470.484,Z 312.013,A -85,B 0,C 180,E1 -7449.296,E2 -7449.296} C_VEL
LIN {X 0,Y 468.064,Z 313.821,A -85,B 0,C 180,E1 -7450.198,E2 -7450.198} C_VEL
LIN {X 0,Y 467.029,Z 315.144,A -85,B 0,C 180,E1 -7450.896,E2 -7450.896} C_VEL
LIN {X 0,Y 466.946,Z 315.566,A -85,B 0,C 180,E1 -7451.134,E2 -7451.134} C_VEL
LIN {X 0,Y 467.003,Z 322.057,A -85,B 0,C 180,E1 -7454.667,E2 -7454.667} C_VEL
LIN {X 0,Y 470.181,Z 336.691,A -85,B 0,C 180,E1 -7455.204,E2 -7455.204} C_VEL
LIN {X 0,Y 470.189,Z 343.934,A -85,B 0,C 180,E1 -7455.501,E2 -7455.501} C_VEL
LIN {X 0,Y 469.803,Z 356.57,A -85,B 0,C 180,E1 -7456.152,E2 -7456.152} C_VEL
LIN {X 0,Y 469.366,Z 367.678,A -85,B 0,C 180,E1 -7456.906,E2 -7456.906} C_VEL
LIN {X 0,Y 468.923,Z 379.009,A -85,B 0,C 180,E1 -7457.888,E2 -7457.888} C_VEL
LIN {X 0,Y 468.438,Z 389.062,A -85,B 0,C 180,E1 -7458.972,E2 -7458.972} C_VEL
LIN {X 0,Y 467.937,Z 398.661,A -85,B 0,C 180,E1 -7460.272,E2 -7460.272} C_VEL
LIN {X 0,Y 467.53,Z 406.378,A -85,B 0,C 180,E1 -7461.572,E2 -7461.572} C_VEL
LIN {X 0,Y 467.271,Z 411.59,A -85,B 0,C 180,E1 -7462.655,E2 -7462.655} C_VEL
LIN {X 0,Y 467.077,Z 416.682,A -85,B 0,C 180,E1 -7463.954,E2 -7463.954} C_VEL
LIN {X 0,Y 466.931,Z 420.626,A -85,B 0,C 180,E1 -7465.251,E2 -7465.251} C_VEL
LIN {X 0,Y 466.858,Z 423.534,A -85,B 0,C 180,E1 -7466.548,E2 -7466.548} C_VEL
LIN {X 0,Y 466.828,Z 424.945,A -85,B 0,C 180,E1 -7467.411,E2 -7467.411} C_VEL
LIN {X 0,Y 466.627,Z 426.557,A -85,B 0,C 180,E1 -7469.137,E2 -7469.137} C_VEL
LIN {X 0,Y 466.613,Z 426.793,A -85,B 0,C 180,E1 -7470,E2 -7470} C_VEL
LIN {X 0,Y 466.699,Z 426.023,A -85,B 0,C 180,E1 -7471.726,E2 -7471.726} C_VEL
LIN {X 0,Y 466.828,Z 425.059,A -85,B 0,C 180,E1 -7472.589,E2 -7472.589} C_VEL
LIN {X 0,Y 466.857,Z 423.709,A -85,B 0,C 180,E1 -7473.452,E2 -7473.452} C_VEL
LIN {X 0,Y 466.912,Z 420.867,A -85,B 0,C 180,E1 -7474.749,E2 -7474.749} C_VEL
LIN {X 0,Y 467.079,Z 417,A -85,B 0,C 180,E1 -7476.046,E2 -7476.046} C_VEL
LIN {X 0,Y 467.272,Z 411.995,A -85,B 0,C 180,E1 -7477.345,E2 -7477.345} C_VEL
LIN {X 0,Y 467.557,Z 405.676,A -85,B 0,C 180,E1 -7478.645,E2 -7478.645} C_VEL
LIN {X 0,Y 467.938,Z 397.82,A -85,B 0,C 180,E1 -7479.946,E2 -7479.946} C_VEL
LIN {X 0,Y 468.454,Z 389.788,A -85,B 0,C 180,E1 -7481.028,E2 -7481.028} C_VEL
LIN {X 0,Y 468.869,Z 379.956,A -85,B 0,C 180,E1 -7482.114,E2 -7482.114} C_VEL
LIN {X 0,Y 469.346,Z 368.799,A -85,B 0,C 180,E1 -7483.096,E2 -7483.096} C_VEL
LIN {X 0,Y 469.793,Z 358.036,A -85,B 0,C 180,E1 -7483.849,E2 -7483.849} C_VEL
LIN {X 0,Y 470.207,Z 345.95,A -85,B 0,C 180,E1 -7484.499,E2 -7484.499} C_VEL
LIN {X 0,Y 470.282,Z 337.227,A -85,B 0,C 180,E1 -7484.863,E2 -7484.863} C_VEL
LIN {X 0,Y 467.628,Z 324.917,A -85,B 0,C 180,E1 -7485.324,E2 -7485.324} C_VEL
LIN {X 0,Y 466.998,Z 322.097,A -85,B 0,C 180,E1 -7485.411,E2 -7485.411} C_VEL
LIN {X 0,Y 466.952,Z 316.34,A -85,B 0,C 180,E1 -7488.521,E2 -7488.521} C_VEL
LIN {X 0,Y 466.981,Z 311.728,A -85,B 0,C 180,E1 -7491.174,E2 -7491.174} C_VEL
LIN {X 0,Y 467.039,Z 307.057,A -85,B 0,C 180,E1 -7493.972,E2 -7493.972} C_VEL
LIN {X 0,Y 467.056,Z 302.379,A -85,B 0,C 180,E1 -7496.835,E2 -7496.835} C_VEL
LIN {X 0,Y 467.106,Z 297.552,A -85,B 0,C 180,E1 -7499.77,E2 -7499.77} C_VEL
LIN {X 0,Y 467.328,Z 291.278,A -85,B 0,C 180,E1 -7503.486,E2 -7503.486} C_VEL
LIN {X 0,Y 467.537,Z 291.251,A -85,B 0,C 180,E1 -7505.891,E2 -7505.891} C_VEL
LIN {X 0,Y 467.585,Z 291.242,A -85,B 0,C 180,E1 -7509.145,E2 -7509.145} C_VEL
LIN {X 0,Y 467.589,Z 291.244,A -85,B 0,C 180,E1 -7512.567,E2 -7512.567} C_VEL
LIN {X 0,Y 467.569,Z 291.247,A -85,B 0,C 180,E1 -7515.053,E2 -7515.053} C_VEL
LIN {X 0,Y 467.592,Z 291.243,A -85,B 0,C 180,E1 -7517.44,E2 -7517.44} C_VEL
LIN {X 0,Y 467.585,Z 291.241,A -85,B 0,C 180,E1 -7520.855,E2 -7520.855} C_VEL
LIN {X 0,Y 467.507,Z 291.253,A -85,B 0,C 180,E1 -7524.106,E2 -7524.106} C_VEL
LIN {X 0,Y 467.273,Z 291.345,A -85,B 0,C 180,E1 -7526.832,E2 -7526.832} C_VEL
LIN {X 0,Y 467.116,Z 297.237,A -85,B 0,C 180,E1 -7530.231,E2 -7530.231} C_VEL
LIN {X 0,Y 467.063,Z 302.304,A -85,B 0,C 180,E1 -7533.165,E2 -7533.165} C_VEL
LIN {X 0,Y 467.046,Z 307.181,A -85,B 0,C 180,E1 -7536.028,E2 -7536.028} C_VEL
LIN {X 0,Y 467.07,Z 312.079,A -85,B 0,C 180,E1 -7538.894,E2 -7538.894} C_VEL
LIN {X 0,Y 466.993,Z 316.638,A -85,B 0,C 180,E1 -7541.576,E2 -7541.576} C_VEL
LIN {X 0,Y 466.994,Z 322.313,A -85,B 0,C 180,E1 -7544.898,E2 -7544.898} C_VEL
LIN {X 0,Y 469.647,Z 335.504,A -85,B 0,C 180,E1 -7545.373,E2 -7545.373} C_VEL
LIN {X 0,Y 469.852,Z 342.35,A -85,B 0,C 180,E1 -7545.656,E2 -7545.656} C_VEL
LIN {X 0,Y 469.442,Z 354.434,A -85,B 0,C 180,E1 -7546.262,E2 -7546.262} C_VEL
LIN {X 0,Y 468.981,Z 367.131,A -85,B 0,C 180,E1 -7547.109,E2 -7547.109} C_VEL
LIN {X 0,Y 468.658,Z 377.581,A -85,B 0,C 180,E1 -7547.991,E2 -7547.991} C_VEL
LIN {X 0,Y 468.184,Z 387.003,A -85,B 0,C 180,E1 -7548.966,E2 -7548.966} C_VEL
LIN {X 0,Y 467.865,Z 395.63,A -85,B 0,C 180,E1 -7550.052,E2 -7550.052} C_VEL
LIN {X 0,Y 467.467,Z 404.078,A -85,B 0,C 180,E1 -7551.353,E2 -7551.353} C_VEL
LIN {X 0,Y 467.246,Z 410.802,A -85,B 0,C 180,E1 -7552.654,E2 -7552.654} C_VEL
LIN {X 0,Y 467.064,Z 416.179,A -85,B 0,C 180,E1 -7553.954,E2 -7553.954} C_VEL
LIN {X 0,Y 466.895,Z 420.363,A -85,B 0,C 180,E1 -7555.251,E2 -7555.251} C_VEL
LIN {X 0,Y 466.857,Z 423.466,A -85,B 0,C 180,E1 -7556.548,E2 -7556.548} C_VEL
LIN {X 0,Y 466.828,Z 425.003,A -85,B 0,C 180,E1 -7557.411,E2 -7557.411} C_VEL
LIN {X 0,Y 466.63,Z 426.761,A -85,B 0,C 180,E1 -7559.137,E2 -7559.137} C_VEL
LIN {X 0,Y 466.617,Z 427.05,A -85,B 0,C 180,E1 -7560,E2 -7560} C_VEL
LIN {X 0,Y 466.631,Z 426.891,A -85,B 0,C 180,E1 -7560.863,E2 -7560.863} C_VEL
LIN {X 0,Y 466.832,Z 425.366,A -85,B 0,C 180,E1 -7562.589,E2 -7562.589} C_VEL
LIN {X 0,Y 466.878,Z 423.965,A -85,B 0,C 180,E1 -7563.452,E2 -7563.452} C_VEL
LIN {X 0,Y 466.923,Z 421.05,A -85,B 0,C 180,E1 -7564.749,E2 -7564.749} C_VEL
LIN {X 0,Y 467.072,Z 417.058,A -85,B 0,C 180,E1 -7566.046,E2 -7566.046} C_VEL
LIN {X 0,Y 467.306,Z 410.908,A -85,B 0,C 180,E1 -7567.562,E2 -7567.562} C_VEL
LIN {X 0,Y 467.59,Z 404.102,A -85,B 0,C 180,E1 -7568.862,E2 -7568.862} C_VEL
LIN {X 0,Y 467.968,Z 395.576,A -85,B 0,C 180,E1 -7570.164,E2 -7570.164} C_VEL
LIN {X 0,Y 468.316,Z 386.819,A -85,B 0,C 180,E1 -7571.25,E2 -7571.25} C_VEL
LIN {X 0,Y 468.856,Z 376.013,A -85,B 0,C 180,E1 -7572.325,E2 -7572.325} C_VEL
LIN {X 0,Y 469.141,Z 365.708,A -85,B 0,C 180,E1 -7573.159,E2 -7573.159} C_VEL
LIN {X 0,Y 469.528,Z 354.903,A -85,B 0,C 180,E1 -7573.857,E2 -7573.857} C_VEL
LIN {X 0,Y 469.914,Z 341.705,A -85,B 0,C 180,E1 -7574.508,E2 -7574.508} C_VEL
LIN {X 0,Y 469.854,Z 336.494,A -85,B 0,C 180,E1 -7574.717,E2 -7574.717} C_VEL
LIN {X 0,Y 467.147,Z 324.101,A -85,B 0,C 180,E1 -7575.212,E2 -7575.212} C_VEL
LIN {X 0,Y 467.155,Z 318.127,A -85,B 0,C 180,E1 -7578.596,E2 -7578.596} C_VEL
LIN {X 0,Y 467.174,Z 313.469,A -85,B 0,C 180,E1 -7581.165,E2 -7581.165} C_VEL
LIN {X 0,Y 467.156,Z 308.198,A -85,B 0,C 180,E1 -7583.966,E2 -7583.966} C_VEL
LIN {X 0,Y 467.13,Z 302.539,A -85,B 0,C 180,E1 -7586.831,E2 -7586.831} C_VEL
LIN {X 0,Y 467.162,Z 296.35,A -85,B 0,C 180,E1 -7589.766,E2 -7589.766} C_VEL
LIN {X 0,Y 467.177,Z 291.296,A -85,B 0,C 180,E1 -7592.025,E2 -7592.025} C_VEL
LIN {X 0,Y 467.526,Z 291.252,A -85,B 0,C 180,E1 -7594.836,E2 -7594.836} C_VEL
LIN {X 0,Y 467.567,Z 291.245,A -85,B 0,C 180,E1 -7598.044,E2 -7598.044} C_VEL
LIN {X 0,Y 467.577,Z 291.243,A -85,B 0,C 180,E1 -7601.276,E2 -7601.276} C_VEL
LIN {X 0,Y 467.551,Z 291.246,A -85,B 0,C 180,E1 -7603.82,E2 -7603.82} C_VEL
LIN {X 0,Y 467.553,Z 291.244,A -85,B 0,C 180,E1 -7606.255,E2 -7606.255} C_VEL
LIN {X 0,Y 467.606,Z 291.295,A -85,B 0,C 180,E1 -7608.384,E2 -7608.384} C_VEL
LIN {X 0,Y 469.293,Z 299.911,A -85,B 0,C 180,E1 -7611.668,E2 -7611.668} C_VEL
LIN {X 0,Y 470.24,Z 305.813,A -85,B 0,C 180,E1 -7613.81,E2 -7613.81} C_VEL
LIN {X 0,Y 469.758,Z 313.598,A -85,B 0,C 180,E1 -7616.389,E2 -7616.389} C_VEL
LIN {X 0,Y 469.298,Z 322.902,A -85,B 0,C 180,E1 -7619.391,E2 -7619.391} C_VEL
LIN {X 0,Y 468.734,Z 333.694,A -85,B 0,C 180,E1 -7622.787,E2 -7622.787} C_VEL
LIN {X 0,Y 468.392,Z 343.049,A -85,B 0,C 180,E1 -7625.63,E2 -7625.63} C_VEL
LIN {X 0,Y 467.956,Z 354.255,A -85,B 0,C 180,E1 -7628.872,E2 -7628.872} C_VEL
LIN {X 0,Y 467.653,Z 365.394,A -85,B 0,C 180,E1 -7632.056,E2 -7632.056} C_VEL
LIN {X 0,Y 467.361,Z 374.329,A -85,B 0,C 180,E1 -7634.575,E2 -7634.575} C_VEL
LIN {X 0,Y 469.693,Z 388.386,A -85,B 0,C 180,E1 -7635.004,E2 -7635.004} C_VEL
LIN {X 0,Y 470.166,Z 393.395,A -85,B 0,C 180,E1 -7635.196,E2 -7635.196} C_VEL
LIN {X 0,Y 469.774,Z 406.18,A -85,B 0,C 180,E1 -7635.764,E2 -7635.764} C_VEL
LIN {X 0,Y 469.257,Z 418.417,A -85,B 0,C 180,E1 -7636.5,E2 -7636.5} C_VEL
LIN {X 0,Y 468.859,Z 428.95,A -85,B 0,C 180,E1 -7637.305,E2 -7637.305} C_VEL
LIN {X 0,Y 468.386,Z 439.592,A -85,B 0,C 180,E1 -7638.313,E2 -7638.313} C_VEL
LIN {X 0,Y 467.877,Z 448.785,A -85,B 0,C 180,E1 -7639.397,E2 -7639.397} C_VEL
LIN {X 0,Y 467.447,Z 457.686,A -85,B 0,C 180,E1 -7640.699,E2 -7640.699} C_VEL
LIN {X 0,Y 467.092,Z 464.848,A -85,B 0,C 180,E1 -7642,E2 -7642} C_VEL
LIN {X 0,Y 466.87,Z 471.224,A -85,B 0,C 180,E1 -7643.479,E2 -7643.479} C_VEL
LIN {X 0,Y 466.784,Z 475.677,A -85,B 0,C 180,E1 -7644.817,E2 -7644.817} C_VEL
LIN {X 0,Y 466.663,Z 477.957,A -85,B 0,C 180,E1 -7645.681,E2 -7645.681} C_VEL
LIN {X 0,Y 466.695,Z 479.806,A -85,B 0,C 180,E1 -7646.547,E2 -7646.547} C_VEL
LIN {X 0,Y 466.646,Z 481.193,A -85,B 0,C 180,E1 -7647.41,E2 -7647.41} C_VEL
LIN {X 0,Y 466.589,Z 482.785,A -85,B 0,C 180,E1 -7649.137,E2 -7649.137} C_VEL
LIN {X 0,Y 466.57,Z 483,A -85,B 0,C 180,E1 -7650,E2 -7650} C_VEL
LIN {X 0,Y 466.589,Z 482.786,A -85,B 0,C 180,E1 -7650.863,E2 -7650.863} C_VEL
LIN {X 0,Y 466.646,Z 481.195,A -85,B 0,C 180,E1 -7652.59,E2 -7652.59} C_VEL
LIN {X 0,Y 466.695,Z 479.81,A -85,B 0,C 180,E1 -7653.453,E2 -7653.453} C_VEL
LIN {X 0,Y 466.703,Z 476.895,A -85,B 0,C 180,E1 -7654.751,E2 -7654.751} C_VEL
LIN {X 0,Y 466.841,Z 472.948,A -85,B 0,C 180,E1 -7656.049,E2 -7656.049} C_VEL
LIN {X 0,Y 466.998,Z 466.875,A -85,B 0,C 180,E1 -7657.567,E2 -7657.567} C_VEL
LIN {X 0,Y 467.35,Z 460.235,A -85,B 0,C 180,E1 -7658.867,E2 -7658.867} C_VEL
LIN {X 0,Y 467.739,Z 451.991,A -85,B 0,C 180,E1 -7660.169,E2 -7660.169} C_VEL
LIN {X 0,Y 468.134,Z 443.517,A -85,B 0,C 180,E1 -7661.254,E2 -7661.254} C_VEL
LIN {X 0,Y 468.66,Z 433.152,A -85,B 0,C 180,E1 -7662.32,E2 -7662.32} C_VEL
LIN {X 0,Y 469.089,Z 421.442,A -85,B 0,C 180,E1 -7663.285,E2 -7663.285} C_VEL
LIN {X 0,Y 469.6,Z 409.039,A -85,B 0,C 180,E1 -7664.075,E2 -7664.075} C_VEL
LIN {X 0,Y 470.089,Z 396.637,A -85,B 0,C 180,E1 -7664.668,E2 -7664.668} C_VEL
LIN {X 0,Y 469.939,Z 390.108,A -85,B 0,C 180,E1 -7664.922,E2 -7664.922} C_VEL
LIN {X 0,Y 467.694,Z 376.685,A -85,B 0,C 180,E1 -7665.364,E2 -7665.364} C_VEL
LIN {X 0,Y 467.34,Z 373.842,A -85,B 0,C 180,E1 -7665.454,E2 -7665.454} C_VEL
LIN {X 0,Y 467.67,Z 361.782,A -85,B 0,C 180,E1 -7668.782,E2 -7668.782} C_VEL
LIN {X 0,Y 467.993,Z 350,A -85,B 0,C 180,E1 -7672.051,E2 -7672.051} C_VEL
LIN {X 0,Y 468.303,Z 340.113,A -85,B 0,C 180,E1 -7674.848,E2 -7674.848} C_VEL
LIN {X 0,Y 468.571,Z 330.102,A -85,B 0,C 180,E1 -7677.757,E2 -7677.757} C_VEL
LIN {X 0,Y 469.017,Z 320.597,A -85,B 0,C 180,E1 -7680.629,E2 -7680.629} C_VEL
LIN {X 0,Y 469.5,Z 309.812,A -85,B 0,C 180,E1 -7684.12,E2 -7684.12} C_VEL
LIN {X 0,Y 469.792,Z 304.149,A -85,B 0,C 180,E1 -7686.115,E2 -7686.115} C_VEL
LIN {X 0,Y 468.947,Z 298.645,A -85,B 0,C 180,E1 -7688.337,E2 -7688.337} C_VEL
LIN {X 0,Y 468.018,Z 293.531,A -85,B 0,C 180,E1 -7690.749,E2 -7690.749} C_VEL
LIN {X 0,Y 467.548,Z 291.249,A -85,B 0,C 180,E1 -7692.128,E2 -7692.128} C_VEL
LIN {X 0,Y 467.567,Z 291.246,A -85,B 0,C 180,E1 -7695.052,E2 -7695.052} C_VEL
LIN {X 0,Y 467.575,Z 291.245,A -85,B 0,C 180,E1 -7698.597,E2 -7698.597} C_VEL
LIN {X 0,Y 467.563,Z 291.244,A -85,B 0,C 180,E1 -7701.409,E2 -7701.409} C_VEL
LIN {X 0,Y 467.562,Z 291.246,A -85,B 0,C 180,E1 -7704.261,E2 -7704.261} C_VEL
LIN {X 0,Y 467.584,Z 291.243,A -85,B 0,C 180,E1 -7707.321,E2 -7707.321} C_VEL
LIN {X 0,Y 467.573,Z 291.244,A -85,B 0,C 180,E1 -7710.667,E2 -7710.667} C_VEL
LIN {X 0,Y 467.589,Z 291.244,A -85,B 0,C 180,E1 -7713.198,E2 -7713.198} C_VEL
LIN {X 0,Y 467.554,Z 291.407,A -85,B 0,C 180,E1 -7715.11,E2 -7715.11} C_VEL
LIN {X 0,Y 467.547,Z 293.677,A -85,B 0,C 180,E1 -7717.927,E2 -7717.927} C_VEL
LIN {X 0,Y 467.506,Z 295.976,A -85,B 0,C 180,E1 -7720.687,E2 -7720.687} C_VEL
LIN {X 0,Y 467.422,Z 298.312,A -85,B 0,C 180,E1 -7723.401,E2 -7723.401} C_VEL
LIN {X 0,Y 467.426,Z 299.656,A -85,B 0,C 180,E1 -7724.926,E2 -7724.926} C_VEL
LIN {X 0,Y 470.22,Z 310.145,A -85,B 0,C 180,E1 -7725.364,E2 -7725.364} C_VEL
LIN {X 0,Y 469.995,Z 323.081,A -85,B 0,C 180,E1 -7725.937,E2 -7725.937} C_VEL
LIN {X 0,Y 469.639,Z 335.113,A -85,B 0,C 180,E1 -7726.647,E2 -7726.647} C_VEL
LIN {X 0,Y 469.233,Z 347.057,A -85,B 0,C 180,E1 -7727.567,E2 -7727.567} C_VEL
LIN {X 0,Y 468.808,Z 357.241,A -85,B 0,C 180,E1 -7728.543,E2 -7728.543} C_VEL
LIN {X 0,Y 468.378,Z 366.394,A -85,B 0,C 180,E1 -7729.627,E2 -7729.627} C_VEL
LIN {X 0,Y 467.981,Z 375.236,A -85,B 0,C 180,E1 -7730.927,E2 -7730.927} C_VEL
LIN {X 0,Y 467.667,Z 382.318,A -85,B 0,C 180,E1 -7732.227,E2 -7732.227} C_VEL
LIN {X 0,Y 467.47,Z 387.907,A -85,B 0,C 180,E1 -7733.526,E2 -7733.526} C_VEL
LIN {X 0,Y 467.194,Z 392.278,A -85,B 0,C 180,E1 -7734.822,E2 -7734.822} C_VEL
LIN {X 0,Y 467.205,Z 394.547,A -85,B 0,C 180,E1 -7735.687,E2 -7735.687} C_VEL
LIN {X 0,Y 467.036,Z 396.404,A -85,B 0,C 180,E1 -7736.549,E2 -7736.549} C_VEL
LIN {X 0,Y 466.88,Z 397.818,A -85,B 0,C 180,E1 -7737.412,E2 -7737.412} C_VEL
LIN {X 0,Y 466.771,Z 399.346,A -85,B 0,C 180,E1 -7739.137,E2 -7739.137} C_VEL
LIN {X 0,Y 466.758,Z 399.524,A -85,B 0,C 180,E1 -7740,E2 -7740} C_VEL
LIN {X 0,Y 466.76,Z 399.271,A -85,B 0,C 180,E1 -7740.863,E2 -7740.863} C_VEL
LIN {X 0,Y 466.86,Z 397.54,A -85,B 0,C 180,E1 -7742.588,E2 -7742.588} C_VEL
LIN {X 0,Y 467.031,Z 396.065,A -85,B 0,C 180,E1 -7743.451,E2 -7743.451} C_VEL
LIN {X 0,Y 467.141,Z 393.02,A -85,B 0,C 180,E1 -7744.746,E2 -7744.746} C_VEL
LIN {X 0,Y 467.227,Z 387.767,A -85,B 0,C 180,E1 -7746.35,E2 -7746.35} C_VEL
LIN {X 0,Y 467.495,Z 381.575,A -85,B 0,C 180,E1 -7747.776,E2 -7747.776} C_VEL
LIN {X 0,Y 467.805,Z 374.435,A -85,B 0,C 180,E1 -7749.076,E2 -7749.076} C_VEL
LIN {X 0,Y 468.153,Z 365.503,A -85,B 0,C 180,E1 -7750.378,E2 -7750.378} C_VEL
LIN {X 0,Y 468.619,Z 356.348,A -85,B 0,C 180,E1 -7751.462,E2 -7751.462} C_VEL
LIN {X 0,Y 469.021,Z 346.235,A -85,B 0,C 180,E1 -7752.439,E2 -7752.439} C_VEL
LIN {X 0,Y 469.357,Z 334.942,A -85,B 0,C 180,E1 -7753.317,E2 -7753.317} C_VEL
LIN {X 0,Y 469.777,Z 322.575,A -85,B 0,C 180,E1 -7754.07,E2 -7754.07} C_VEL
LIN {X 0,Y 470.07,Z 309.208,A -85,B 0,C 180,E1 -7754.669,E2 -7754.669} C_VEL
LIN {X 0,Y 466.989,Z 295.886,A -85,B 0,C 180,E1 -7755.209,E2 -7755.209} C_VEL
LIN {X 0,Y 466.942,Z 292.013,A -85,B 0,C 180,E1 -7758.518,E2 -7758.518} C_VEL
LIN {X 0,Y 466.95,Z 291.323,A -85,B 0,C 180,E1 -7759.337,E2 -7759.337} C_VEL
LIN {X 0,Y 467.245,Z 291.284,A -85,B 0,C 180,E1 -7762.088,E2 -7762.088} C_VEL
LIN {X 0,Y 467.524,Z 291.248,A -85,B 0,C 180,E1 -7764.892,E2 -7764.892} C_VEL
LIN {X 0,Y 467.619,Z 291.231,A -85,B 0,C 180,E1 -7767.769,E2 -7767.769} C_VEL
LIN {X 0,Y 467.57,Z 291.237,A -85,B 0,C 180,E1 -7771.045,E2 -7771.045} C_VEL
LIN {X 0,Y 467.592,Z 291.243,A -85,B 0,C 180,E1 -7774.242,E2 -7774.242} C_VEL
LIN {X 0,Y 467.551,Z 291.243,A -85,B 0,C 180,E1 -7777.186,E2 -7777.186} C_VEL
LIN {X 0,Y 467.58,Z 291.245,A -85,B 0,C 180,E1 -7780.265,E2 -7780.265} C_VEL
LIN {X 0,Y 467.589,Z 291.24,A -85,B 0,C 180,E1 -7782.567,E2 -7782.567} C_VEL
LIN {X 0,Y 467.573,Z 291.239,A -85,B 0,C 180,E1 -7785.053,E2 -7785.053} C_VEL
LIN {X 0,Y 467.592,Z 291.239,A -85,B 0,C 180,E1 -7787.44,E2 -7787.44} C_VEL
LIN {X 0,Y 467.585,Z 291.238,A -85,B 0,C 180,E1 -7790.855,E2 -7790.855} C_VEL
LIN {X 0,Y 467.536,Z 291.247,A -85,B 0,C 180,E1 -7794.265,E2 -7794.265} C_VEL
LIN {X 0,Y 467.318,Z 291.412,A -85,B 0,C 180,E1 -7796.707,E2 -7796.707} C_VEL
LIN {X 0,Y 467.102,Z 297.384,A -85,B 0,C 180,E1 -7800.23,E2 -7800.23} C_VEL
LIN {X 0,Y 467.055,Z 302.212,A -85,B 0,C 180,E1 -7803.165,E2 -7803.165} C_VEL
LIN {X 0,Y 467.038,Z 306.897,A -85,B 0,C 180,E1 -7806.027,E2 -7806.027} C_VEL
LIN {X 0,Y 467.011,Z 311.722,A -85,B 0,C 180,E1 -7808.913,E2 -7808.913} C_VEL
LIN {X 0,Y 466.946,Z 315.566,A -85,B 0,C 180,E1 -7811.134,E2 -7811.134} C_VEL
LIN {X 0,Y 466.263,Z 316.47,A -85,B 0,C 180,E1 -7811.601,E2 -7811.601} C_VEL
LIN {X 0,Y 463.395,Z 318.094,A -85,B 0,C 180,E1 -7812.324,E2 -7812.324} C_VEL
LIN {X 0,Y 460.523,Z 319.751,A -85,B 0,C 180,E1 -7813.055,E2 -7813.055} C_VEL
LIN {X 0,Y 459.853,Z 320.715,A -85,B 0,C 180,E1 -7813.53,E2 -7813.53} C_VEL
LIN {X 0,Y 459.934,Z 322.568,A -85,B 0,C 180,E1 -7814.447,E2 -7814.447} C_VEL
LIN {X 0,Y 462.891,Z 335.588,A -85,B 0,C 180,E1 -7814.913,E2 -7814.913} C_VEL
LIN {X 0,Y 463.482,Z 339.706,A -85,B 0,C 180,E1 -7815.09,E2 -7815.09} C_VEL
LIN {X 0,Y 463.148,Z 352.192,A -85,B 0,C 180,E1 -7815.668,E2 -7815.668} C_VEL
LIN {X 0,Y 462.703,Z 363.215,A -85,B 0,C 180,E1 -7816.349,E2 -7816.349} C_VEL
LIN {X 0,Y 462.229,Z 374.72,A -85,B 0,C 180,E1 -7817.264,E2 -7817.264} C_VEL
LIN {X 0,Y 461.762,Z 384.721,A -85,B 0,C 180,E1 -7818.254,E2 -7818.254} C_VEL
LIN {X 0,Y 461.285,Z 392.931,A -85,B 0,C 180,E1 -7819.243,E2 -7819.243} C_VEL
LIN {X 0,Y 460.882,Z 400.507,A -85,B 0,C 180,E1 -7820.344,E2 -7820.344} C_VEL
LIN {X 0,Y 460.468,Z 407.893,A -85,B 0,C 180,E1 -7821.663,E2 -7821.663} C_VEL
LIN {X 0,Y 460.119,Z 414.448,A -85,B 0,C 180,E1 -7823.137,E2 -7823.137} C_VEL
LIN {X 0,Y 459.897,Z 418.517,A -85,B 0,C 180,E1 -7824.299,E2 -7824.299} C_VEL
LIN {X 0,Y 459.897,Z 422.098,A -85,B 0,C 180,E1 -7825.618,E2 -7825.618} C_VEL
LIN {X 0,Y 459.793,Z 423.949,A -85,B 0,C 180,E1 -7826.495,E2 -7826.495} C_VEL
LIN {X 0,Y 459.756,Z 425.36,A -85,B 0,C 180,E1 -7827.372,E2 -7827.372} C_VEL
LIN {X 0,Y 459.56,Z 426.971,A -85,B 0,C 180,E1 -7829.124,E2 -7829.124} C_VEL
LIN {X 0,Y 459.544,Z 427.207,A -85,B 0,C 180,E1 -7830,E2 -7830} C_VEL
LIN {X 0,Y 459.639,Z 426.436,A -85,B 0,C 180,E1 -7831.752,E2 -7831.752} C_VEL
LIN {X 0,Y 459.756,Z 425.472,A -85,B 0,C 180,E1 -7832.628,E2 -7832.628} C_VEL
LIN {X 0,Y 459.791,Z 424.122,A -85,B 0,C 180,E1 -7833.505,E2 -7833.505} C_VEL
LIN {X 0,Y 459.835,Z 421.28,A -85,B 0,C 180,E1 -7834.822,E2 -7834.822} C_VEL
LIN {X 0,Y 460.04,Z 417.411,A -85,B 0,C 180,E1 -7836.139,E2 -7836.139} C_VEL
LIN {X 0,Y 460.244,Z 412.405,A -85,B 0,C 180,E1 -7837.458,E2 -7837.458} C_VEL
LIN {X 0,Y 460.565,Z 406.084,A -85,B 0,C 180,E1 -7838.777,E2 -7838.777} C_VEL
LIN {X 0,Y 460.964,Z 398.226,A -85,B 0,C 180,E1 -7840.098,E2 -7840.098} C_VEL
LIN {X 0,Y 461.496,Z 390.193,A -85,B 0,C 180,E1 -7841.196,E2 -7841.196} C_VEL
LIN {X 0,Y 461.953,Z 380.354,A -85,B 0,C 180,E1 -7842.298,E2 -7842.298} C_VEL
LIN {X 0,Y 462.446,Z 368.922,A -85,B 0,C 180,E1 -7843.317,E2 -7843.317} C_VEL
LIN {X 0,Y 462.911,Z 358.423,A -85,B 0,C 180,E1 -7844.059,E2 -7844.059} C_VEL
LIN {X 0,Y 463.356,Z 346.321,A -85,B 0,C 180,E1 -7844.718,E2 -7844.718} C_VEL
LIN {X 0,Y 463.412,Z 338.232,A -85,B 0,C 180,E1 -7845.063,E2 -7845.063} C_VEL
LIN {X 0,Y 460.672,Z 325.55,A -85,B 0,C 180,E1 -7845.555,E2 -7845.555} C_VEL
LIN {X 0,Y 459.936,Z 322.432,A -85,B 0,C 180,E1 -7845.657,E2 -7845.657} C_VEL
LIN {X 0,Y 459.888,Z 316.772,A -85,B 0,C 180,E1 -7848.719,E2 -7848.719} C_VEL
LIN {X 0,Y 459.941,Z 311.921,A -85,B 0,C 180,E1 -7851.514,E2 -7851.514} C_VEL
LIN {X 0,Y 459.986,Z 307.189,A -85,B 0,C 180,E1 -7854.364,E2 -7854.364} C_VEL
LIN {X 0,Y 460.029,Z 301.874,A -85,B 0,C 180,E1 -7857.614,E2 -7857.614} C_VEL
LIN {X 0,Y 460.074,Z 297.519,A -85,B 0,C 180,E1 -7860.272,E2 -7860.272} C_VEL
LIN {X 0,Y 460.271,Z 292.157,A -85,B 0,C 180,E1 -7863.477,E2 -7863.477} C_VEL
LIN {X 0,Y 460.483,Z 292.129,A -85,B 0,C 180,E1 -7866.011,E2 -7866.011} C_VEL
LIN {X 0,Y 460.547,Z 292.119,A -85,B 0,C 180,E1 -7868.898,E2 -7868.898} C_VEL
LIN {X 0,Y 460.526,Z 292.122,A -85,B 0,C 180,E1 -7872.181,E2 -7872.181} C_VEL
LIN {X 0,Y 460.516,Z 292.123,A -85,B 0,C 180,E1 -7875.411,E2 -7875.411} C_VEL
LIN {X 0,Y 460.535,Z 292.119,A -85,B 0,C 180,E1 -7878.398,E2 -7878.398} C_VEL
LIN {X 0,Y 460.528,Z 292.121,A -85,B 0,C 180,E1 -7881.267,E2 -7881.267} C_VEL
LIN {X 0,Y 460.447,Z 292.129,A -85,B 0,C 180,E1 -7884.548,E2 -7884.548} C_VEL
LIN {X 0,Y 460.218,Z 292.329,A -85,B 0,C 180,E1 -7886.933,E2 -7886.933} C_VEL
LIN {X 0,Y 460.085,Z 298.875,A -85,B 0,C 180,E1 -7890.737,E2 -7890.737} C_VEL
LIN {X 0,Y 460.014,Z 303.962,A -85,B 0,C 180,E1 -7893.701,E2 -7893.701} C_VEL
LIN {X 0,Y 459.978,Z 308.891,A -85,B 0,C 180,E1 -7896.593,E2 -7896.593} C_VEL
LIN {X 0,Y 459.95,Z 313.668,A -85,B 0,C 180,E1 -7899.425,E2 -7899.425} C_VEL
LIN {X 0,Y 459.885,Z 318.417,A -85,B 0,C 180,E1 -7902.203,E2 -7902.203} C_VEL
LIN {X 0,Y 459.944,Z 322.841,A -85,B 0,C 180,E1 -7904.697,E2 -7904.697} C_VEL
LIN {X 0,Y 462.699,Z 336.221,A -85,B 0,C 180,E1 -7905.19,E2 -7905.19} C_VEL
LIN {X 0,Y 462.972,Z 340.796,A -85,B 0,C 180,E1 -7905.382,E2 -7905.382} C_VEL
LIN {X 0,Y 462.534,Z 354.112,A -85,B 0,C 180,E1 -7906.042,E2 -7906.042} C_VEL
LIN {X 0,Y 462.069,Z 365.8,A -85,B 0,C 180,E1 -7906.812,E2 -7906.812} C_VEL
LIN {X 0,Y 461.745,Z 376.443,A -85,B 0,C 180,E1 -7907.697,E2 -7907.697} C_VEL
LIN {X 0,Y 461.316,Z 385.192,A -85,B 0,C 180,E1 -7908.577,E2 -7908.577} C_VEL
LIN {X 0,Y 460.942,Z 394.259,A -85,B 0,C 180,E1 -7909.68,E2 -7909.68} C_VEL
LIN {X 0,Y 460.523,Z 403.023,A -85,B 0,C 180,E1 -7911.001,E2 -7911.001} C_VEL
LIN {X 0,Y 460.238,Z 410.102,A -85,B 0,C 180,E1 -7912.321,E2 -7912.321} C_VEL
LIN {X 0,Y 460.081,Z 415.112,A -85,B 0,C 180,E1 -7913.481,E2 -7913.481} C_VEL
LIN {X 0,Y 459.779,Z 419.482,A -85,B 0,C 180,E1 -7914.738,E2 -7914.738} C_VEL
LIN {X 0,Y 459.885,Z 421.892,A -85,B 0,C 180,E1 -7915.618,E2 -7915.618} C_VEL
LIN {X 0,Y 459.792,Z 423.862,A -85,B 0,C 180,E1 -7916.495,E2 -7916.495} C_VEL
LIN {X 0,Y 459.756,Z 425.414,A -85,B 0,C 180,E1 -7917.371,E2 -7917.371} C_VEL
LIN {X 0,Y 459.64,Z 426.505,A -85,B 0,C 180,E1 -7918.248,E2 -7918.248} C_VEL
LIN {X 0,Y 459.547,Z 427.495,A -85,B 0,C 180,E1 -7920,E2 -7920} C_VEL
LIN {X 0,Y 459.564,Z 427.346,A -85,B 0,C 180,E1 -7920.876,E2 -7920.876} C_VEL
LIN {X 0,Y 459.777,Z 425.833,A -85,B 0,C 180,E1 -7922.628,E2 -7922.628} C_VEL
LIN {X 0,Y 459.81,Z 424.441,A -85,B 0,C 180,E1 -7923.505,E2 -7923.505} C_VEL
LIN {X 0,Y 459.865,Z 421.528,A -85,B 0,C 180,E1 -7924.822,E2 -7924.822} C_VEL
LIN {X 0,Y 460.034,Z 417.531,A -85,B 0,C 180,E1 -7926.139,E2 -7926.139} C_VEL
LIN {X 0,Y 460.3,Z 411.368,A -85,B 0,C 180,E1 -7927.678,E2 -7927.678} C_VEL
LIN {X 0,Y 460.604,Z 404.544,A -85,B 0,C 180,E1 -7928.998,E2 -7928.998} C_VEL
LIN {X 0,Y 461.002,Z 395.999,A -85,B 0,C 180,E1 -7930.319,E2 -7930.319} C_VEL
LIN {X 0,Y 461.456,Z 386.24,A -85,B 0,C 180,E1 -7931.531,E2 -7931.531} C_VEL
LIN {X 0,Y 461.969,Z 375.493,A -85,B 0,C 180,E1 -7932.602,E2 -7932.602} C_VEL
LIN {X 0,Y 462.314,Z 364.516,A -85,B 0,C 180,E1 -7933.477,E2 -7933.477} C_VEL
LIN {X 0,Y 462.794,Z 351.448,A -85,B 0,C 180,E1 -7934.287,E2 -7934.287} C_VEL
LIN {X 0,Y 463.075,Z 338.063,A -85,B 0,C 180,E1 -7934.896,E2 -7934.896} C_VEL
LIN {X 0,Y 460.473,Z 326.224,A -85,B 0,C 180,E1 -7935.379,E2 -7935.379} C_VEL
LIN {X 0,Y 460.124,Z 324.655,A -85,B 0,C 180,E1 -7935.439,E2 -7935.439} C_VEL
LIN {X 0,Y 460.137,Z 318.839,A -85,B 0,C 180,E1 -7938.742,E2 -7938.742} C_VEL
LIN {X 0,Y 460.133,Z 313.806,A -85,B 0,C 180,E1 -7941.504,E2 -7941.504} C_VEL
LIN {X 0,Y 460.117,Z 308.434,A -85,B 0,C 180,E1 -7944.356,E2 -7944.356} C_VEL
LIN {X 0,Y 460.1,Z 301.916,A -85,B 0,C 180,E1 -7947.631,E2 -7947.631} C_VEL
LIN {X 0,Y 460.122,Z 296.247,A -85,B 0,C 180,E1 -7950.268,E2 -7950.268} C_VEL
LIN {X 0,Y 460.163,Z 292.17,A -85,B 0,C 180,E1 -7952.12,E2 -7952.12} C_VEL
LIN {X 0,Y 460.468,Z 292.13,A -85,B 0,C 180,E1 -7954.493,E2 -7954.493} C_VEL
LIN {X 0,Y 460.503,Z 292.125,A -85,B 0,C 180,E1 -7957.623,E2 -7957.623} C_VEL
LIN {X 0,Y 460.538,Z 292.122,A -85,B 0,C 180,E1 -7960.269,E2 -7960.269} C_VEL
LIN {X 0,Y 460.512,Z 292.124,A -85,B 0,C 180,E1 -7963.374,E2 -7963.374} C_VEL
LIN {X 0,Y 460.512,Z 292.122,A -85,B 0,C 180,E1 -7966.626,E2 -7966.626} C_VEL
LIN {X 0,Y 460.546,Z 292.227,A -85,B 0,C 180,E1 -7968.063,E2 -7968.063} C_VEL
LIN {X 0,Y 461.983,Z 299.481,A -85,B 0,C 180,E1 -7970.882,E2 -7970.882} C_VEL
LIN {X 0,Y 463.221,Z 306.606,A -85,B 0,C 180,E1 -7973.525,E2 -7973.525} C_VEL
LIN {X 0,Y 462.953,Z 313.332,A -85,B 0,C 180,E1 -7975.827,E2 -7975.827} C_VEL
LIN {X 0,Y 462.309,Z 324.179,A -85,B 0,C 180,E1 -7979.385,E2 -7979.385} C_VEL
LIN {X 0,Y 461.708,Z 334.97,A -85,B 0,C 180,E1 -7982.829,E2 -7982.829} C_VEL
LIN {X 0,Y 461.303,Z 345.534,A -85,B 0,C 180,E1 -7986.08,E2 -7986.08} C_VEL
LIN {X 0,Y 460.833,Z 357.092,A -85,B 0,C 180,E1 -7989.466,E2 -7989.466} C_VEL
LIN {X 0,Y 460.467,Z 368.214,A -85,B 0,C 180,E1 -7992.685,E2 -7992.685} C_VEL
LIN {X 0,Y 460.328,Z 374.08,A -85,B 0,C 180,E1 -7994.332,E2 -7994.332} C_VEL
LIN {X 0,Y 462.594,Z 387.867,A -85,B 0,C 180,E1 -7994.767,E2 -7994.767} C_VEL
LIN {X 0,Y 463.268,Z 393.724,A -85,B 0,C 180,E1 -7995.002,E2 -7995.002} C_VEL
LIN {X 0,Y 462.825,Z 406.63,A -85,B 0,C 180,E1 -7995.602,E2 -7995.602} C_VEL
LIN {X 0,Y 462.273,Z 418.959,A -85,B 0,C 180,E1 -7996.37,E2 -7996.37} C_VEL
LIN {X 0,Y 461.832,Z 429.018,A -85,B 0,C 180,E1 -7997.165,E2 -7997.165} C_VEL
LIN {X 0,Y 461.4,Z 439.001,A -85,B 0,C 180,E1 -7998.134,E2 -7998.134} C_VEL
LIN {X 0,Y 460.829,Z 448.246,A -85,B 0,C 180,E1 -7999.233,E2 -7999.233} C_VEL
LIN {X 0,Y 460.396,Z 457.272,A -85,B 0,C 180,E1 -8000.555,E2 -8000.555} C_VEL
LIN {X 0,Y 460.055,Z 464.544,A -85,B 0,C 180,E1 -8001.876,E2 -8001.876} C_VEL
LIN {X 0,Y 459.848,Z 469.458,A -85,B 0,C 180,E1 -8002.977,E2 -8002.977} C_VEL
LIN {X 0,Y 459.756,Z 474.244,A -85,B 0,C 180,E1 -8004.298,E2 -8004.298} C_VEL
LIN {X 0,Y 459.58,Z 477.892,A -85,B 0,C 180,E1 -8005.615,E2 -8005.615} C_VEL
LIN {X 0,Y 459.591,Z 479.773,A -85,B 0,C 180,E1 -8006.493,E2 -8006.493} C_VEL
LIN {X 0,Y 459.57,Z 481.176,A -85,B 0,C 180,E1 -8007.37,E2 -8007.37} C_VEL
LIN {X 0,Y 459.494,Z 482.779,A -85,B 0,C 180,E1 -8009.124,E2 -8009.124} C_VEL
LIN {X 0,Y 459.474,Z 482.994,A -85,B 0,C 180,E1 -8010,E2 -8010} C_VEL
LIN {X 0,Y 459.494,Z 482.779,A -85,B 0,C 180,E1 -8010.876,E2 -8010.876} C_VEL
LIN {X 0,Y 459.57,Z 481.178,A -85,B 0,C 180,E1 -8012.63,E2 -8012.63} C_VEL
LIN {X 0,Y 459.591,Z 479.777,A -85,B 0,C 180,E1 -8013.507,E2 -8013.507} C_VEL
LIN {X 0,Y 459.635,Z 476.812,A -85,B 0,C 180,E1 -8014.824,E2 -8014.824} C_VEL
LIN {X 0,Y 459.758,Z 472.78,A -85,B 0,C 180,E1 -8016.143,E2 -8016.143} C_VEL
LIN {X 0,Y 459.929,Z 466.57,A -85,B 0,C 180,E1 -8017.684,E2 -8017.684} C_VEL
LIN {X 0,Y 460.284,Z 459.797,A -85,B 0,C 180,E1 -8019.004,E2 -8019.004} C_VEL
LIN {X 0,Y 460.677,Z 451.388,A -85,B 0,C 180,E1 -8020.326,E2 -8020.326} C_VEL
LIN {X 0,Y 461.137,Z 442.774,A -85,B 0,C 180,E1 -8021.428,E2 -8021.428} C_VEL
LIN {X 0,Y 461.645,Z 432.525,A -85,B 0,C 180,E1 -8022.494,E2 -8022.494} C_VEL
LIN {X 0,Y 462.069,Z 421.639,A -85,B 0,C 180,E1 -8023.412,E2 -8023.412} C_VEL
LIN {X 0,Y 462.586,Z 410.184,A -85,B 0,C 180,E1 -8024.181,E2 -8024.181} C_VEL
LIN {X 0,Y 463.096,Z 398.473,A -85,B 0,C 180,E1 -8024.782,E2 -8024.782} C_VEL
LIN {X 0,Y 463.133,Z 391.84,A -85,B 0,C 180,E1 -8025.056,E2 -8025.056} C_VEL
LIN {X 0,Y 460.943,Z 378.182,A -85,B 0,C 180,E1 -8025.549,E2 -8025.549} C_VEL
LIN {X 0,Y 460.268,Z 373.147,A -85,B 0,C 180,E1 -8025.686,E2 -8025.686} C_VEL
LIN {X 0,Y 460.59,Z 361.697,A -85,B 0,C 180,E1 -8028.908,E2 -8028.908} C_VEL
LIN {X 0,Y 460.905,Z 350.976,A -85,B 0,C 180,E1 -8031.936,E2 -8031.936} C_VEL
LIN {X 0,Y 461.228,Z 341.12,A -85,B 0,C 180,E1 -8034.774,E2 -8034.774} C_VEL
LIN {X 0,Y 461.511,Z 331.643,A -85,B 0,C 180,E1 -8037.578,E2 -8037.578} C_VEL
LIN {X 0,Y 461.997,Z 321.73,A -85,B 0,C 180,E1 -8040.638,E2 -8040.638} C_VEL
LIN {X 0,Y 462.55,Z 310.976,A -85,B 0,C 180,E1 -8044.207,E2 -8044.207} C_VEL
LIN {X 0,Y 462.803,Z 304.953,A -85,B 0,C 180,E1 -8046.405,E2 -8046.405} C_VEL
LIN {X 0,Y 461.79,Z 298.676,A -85,B 0,C 180,E1 -8049.088,E2 -8049.088} C_VEL
LIN {X 0,Y 460.817,Z 293.747,A -85,B 0,C 180,E1 -8051.642,E2 -8051.642} C_VEL
LIN {X 0,Y 460.505,Z 292.127,A -85,B 0,C 180,E1 -8052.737,E2 -8052.737} C_VEL
LIN {X 0,Y 460.507,Z 292.125,A -85,B 0,C 180,E1 -8055.831,E2 -8055.831} C_VEL
LIN {X 0,Y 460.53,Z 292.121,A -85,B 0,C 180,E1 -8058.988,E2 -8058.988} C_VEL
LIN {X 0,Y 460.521,Z 292.122,A -85,B 0,C 180,E1 -8061.266,E2 -8061.266} C_VEL
LIN {X 0,Y 460.513,Z 292.123,A -85,B 0,C 180,E1 -8064.554,E2 -8064.554} C_VEL
LIN {X 0,Y 460.534,Z 292.122,A -85,B 0,C 180,E1 -8067.716,E2 -8067.716} C_VEL
LIN {X 0,Y 460.543,Z 292.12,A -85,B 0,C 180,E1 -8070.769,E2 -8070.769} C_VEL
LIN {X 0,Y 460.54,Z 292.122,A -85,B 0,C 180,E1 -8073.733,E2 -8073.733} C_VEL
LIN {X 0,Y 460.529,Z 292.335,A -85,B 0,C 180,E1 -8074.704,E2 -8074.704} C_VEL
LIN {X 0,Y 460.589,Z 293.828,A -85,B 0,C 180,E1 -8076.626,E2 -8076.626} C_VEL
LIN {X 0,Y 460.563,Z 296.099,A -85,B 0,C 180,E1 -8079.453,E2 -8079.453} C_VEL
LIN {X 0,Y 460.462,Z 298.416,A -85,B 0,C 180,E1 -8082.226,E2 -8082.226} C_VEL
LIN {X 0,Y 460.435,Z 300.531,A -85,B 0,C 180,E1 -8084.678,E2 -8084.678} C_VEL
LIN {X 0,Y 463.44,Z 311.732,A -85,B 0,C 180,E1 -8085.173,E2 -8085.173} C_VEL
LIN {X 0,Y 463.108,Z 324.98,A -85,B 0,C 180,E1 -8085.779,E2 -8085.779} C_VEL
LIN {X 0,Y 462.781,Z 336.103,A -85,B 0,C 180,E1 -8086.458,E2 -8086.458} C_VEL
LIN {X 0,Y 462.346,Z 347.863,A -85,B 0,C 180,E1 -8087.378,E2 -8087.378} C_VEL
LIN {X 0,Y 461.895,Z 358.025,A -85,B 0,C 180,E1 -8088.369,E2 -8088.369} C_VEL
LIN {X 0,Y 461.445,Z 367.154,A -85,B 0,C 180,E1 -8089.469,E2 -8089.469} C_VEL
LIN {X 0,Y 461.027,Z 375.972,A -85,B 0,C 180,E1 -8090.789,E2 -8090.789} C_VEL
LIN {X 0,Y 460.668,Z 383.054,A -85,B 0,C 180,E1 -8092.108,E2 -8092.108} C_VEL
